FUNCTION "CWA_ScaleCtrlSub" : VOID	// FC 40
TITLE = CWA SUBROUTINE
//  
//COPYRIGHT:    (C) 1996 BY  BUHLER LTD.
//                           CH-9240 UZWIL  SWITZERLAND
//
//PRODUCT:      CWA
//
//TITLE:        SCALE CONTROL: SUBROUTINE
//
//-------------------------------------------------------------------------
//
//IDENT:        AUTOR:              DEPT:                         DATE:
//
//FC40.1.8      A. Egli             CT3                           27-Jun-2005
//              Working step: Do not calculate ingredient size 
//FC40.1.7      A. Egli             CT3                           21-Sep-2004
//              Registration: Test Ingr.WtActual >0 
//FC40.1.6      A. Egli             CT3                           12-Jun-2003
//              Test if more than 48 bins 
//FC40.1.5      A. Egli             CT3                           12-April-2000
//              Negativ CutoffWt >= 2* ParTolPosWt 
//FC40.1E       A. Egli             CT3                           12-Nov-98
//              Fault in SUBROUTINE EMPTYING_MONITORING 
//              Run closing delay only if scale is open
//FC40.1D       A. Egli             CT3                           24-Jun-98
//              Start part recipe
//              DBB52: First Ingredient
//              DBB53: Number of Ingredient
//FC40.1C       A. Egli             AEE61                         18-Mar-98
//              Update to S5 Version 2F
//
//FC40.1B       A. Egli             AEE61                         20-Jan-98
//              Update to S5 Version 2D
//
//FC40.1A       S. Kalberer         AEE61                         24-Apr-96
//              1st Release in S7, converted from FB40.1D
//
//-------------------------------------------------------------------------
//
//PURPOSE:      MANUAL : CWAMAN
//
//RESTRICTIONS:
//
//-------------------------------------------------------------------------
//
//$EJECT
//
AUTHOR : EA
FAMILY : CWA
NAME : CWASubr
VERSION : 1.8
VAR_TEMP
  InCode : WORD ;	//InFunctionCode
  TargetAddress : DWORD ;	//temp address pointer
  Cnt : WORD ;	//temp loop counter
  tmpAddr : DWORD ;
  tmpTimeTarget : INT ;
  tmpTimeTotal : INT ;
  tmpWtPartIngr : DINT ;
  tmpWtDiff : DINT ;
  tmpWtCorr : DINT ;
  tmpWt : DINT ;
  tmpBinNr : INT ;
  tmpWtDiffIsPos : BOOL ;
END_VAR
BEGIN
NETWORK
TITLE = FC-PARAMETER
//FC-PARAMETER:
//-------------
//  CODE: CODE OF EXECUTING FUNCTION
//        KY 0,0   : SUBROUTINE RESET TIMER
//        KY 0,1   : SUBROUTINE RUN DosingMonDelay
//        KY 0,2   : SUBROUTINE RUN SettlingTime
//        KY 0,4   : SUBROUTINE DOSING_MONITORING
//        KY 0,5   : SUBROUTINE EMPTYING_MONITORING
//        KY 0,8   : SUBROUTINE RUN DAMPENING TIME SCALE CLOSED
//        KY 0,10  : SUBROUTINE RUN CLOSING DELAY IF EMPTY
//        KY 0,11  : SUBROUTINE CORRECTION CUTOFF VALUE
//        KY 0,12  : SUBROUTINE TOLERANCE TEST
//                   Input : DW196 = var_tol._pos_unit
//                           DW197 = var_tol._pos_%
//                   Output: M199.0: 1=fault pos
//                   Output: M199.1: 1=fault neg
//                   Output: M199.2: 1=Ingr.Done
//        KY 1,1   : SUBROUTINE TEST_RESULT_DB
//        KY 1,2   : SUBROUTINE INIT_RESULT
//        KY 1,4   : SUBROUTINE REGISTRATION_INGREDIENT
//        KY 2,1   : SUBROUTINE TEST_RECIPE_DB
//        KY 2,2   : SUBROUTINE COUNT INGR
//        KY 2,4   : SUBROUTINE READ RECIPE INGR
//        KY 2,8   : SUBROUTINE MODIFY_RECIPE
//        KY 4,1   : SUBROUTINE TEST_BIN_PARAMETER_DB
//        KY 4,2   : SUBROUTINE READ_BIN_PARA
//        KY 4,4   : SUBROUTINE WRITE_BIN_PARA
//        KY 4,8   : SUBROUTINE TEST BIN
//                      Input  : DW195 = Bin-Nr
//                      Output : M 199.3 : 1= Fault
//                               DW197 = DW_NR_Bin
//                               DW198 = relBinNr
//
//ACTUAL DB BY CALL: SCALE    DB
//AUFGESCHALGENER  : WAAGEN   DB
//
//
      T     #InCode;
NETWORK
TITLE = Subroutine Reset Time
//Not implemented.
//Instead of this function call, write your self:
//      L     S5T#0MS                     // Partimer_1
//      SE    T [DBW 24]                  // --> Reset Timer
NETWORK
TITLE =  Subroutine Run DosingMonDelay
      L     #InCode;
      L     B#(0, 1);	// CODE= Run Settling time dos.
      <>I;
      JC    NX4;	// NEXT;
      AN    M 189.3;	// --> inf_DelayMon
      ON    "SYS_Tick1s";
      BEC;
      L     DBW 96;	// var_DosingMonDelay
      +     10;
      T     DBW 96;	// var_DosingMonDelay
      L     DBW 160;	// ParDosingMonDelay
      >=I;
      R     M 189.3;	// --> inf_DelayMon
      BEU;
NETWORK
TITLE =  Subroutine Run Settling time
NX4:  L     #InCode;
      L     B#(0, 2);	// CODE= Run Settling time
      <>I;
      JC    NX5;
      L     W#16#999;
      L     DBW 194;	// ParSettlingTime
      DTB;
      <D;
      JC    NX4s;
      L     W#16#1000;	// time_base 1/10s
NX4a: OW;
      A     M 193.4;	// --> sta_SettlingTime
      SD    T [DBW 24];	// Partimer_1 --> Timer
      A     T [DBW 24];	// Partimer_1 --> Timer
      R     M 193.4;	// --> sta_SettlingTime
      BEU;
NX4s: SRW   4;
      L     W#16#2000;	// time_base 1 s
      JU    NX4a;
NETWORK
TITLE =  Subroutine Dosing monitoring
NX5:  L     #InCode;
      L     B#(0, 4);	// CODE= dos_MONITORING
      <>I;
      JC    NX6;	// NEXT;
      L     DBW 378;	// var_MonTime
      L     0;
      >I;
      JC    OK5;	// -- INIT --------------------
      L     DBW 162;	// ParDosingMonTime
      T     DBW 378;	// --> var_MonTime
      L     DBD 254;	// inf_ScaleWt
      T     DBD 380;	// --> var_MonTara
OK5:  AN    "SYS_Tick1s";	// -- CONTROL -----------------
      BEC;
      A     M 191.2;	// es_DosingMon
      O     M 189.3;	// inf_DosingMon
      JC    TI2;
      L     DBW 378;	// var_MonTime [1/10s]
      +     -10;
      T     DBW 378;	// --> var_MonTime [1/10s]
      L     0;
      >I;
      JC    TI2;	// --- CONTROL ---------------
      L     DBW 166;	// ParDosingMonWtFast
      A     M 180.6;	// outp_DosingFast
      JC    X1;
      L     DBW 168;	// ParDosingMinWtSlow
X1:   L     DBD 380;	// var_MonTara
      A     DBX 7.0;	// ParNegativeWeighing
      JC    NX5n;
      +D;
      L     DBD 254;	// inf_ScaleWt
      >=D;
      AN    DBX 7.0;	// ParNegativeWeighing
      JC    ERRO;
      JU    TI2;
NX5n: TAK;
      -D;
      L     DBD 254;	// inf_ScaleWt
      <D;
      JC    ERRO;
      JU    TI2;
ERRO: S     M 191.2;	// --> es_time_outdos
      L     63;
      T     DBW 246;	// --> errCodeSW
TI2:  L     DBW 328;	// Ingr.DosingTime
      L     DBW 354;	// ParDosingTimeMax
      <=I;
      O(;
      L     0;	// no monitioring
      ==I;
      );
      BEC;	// --- error 2 -------------------
      S     M 191.4;	// --> es_DosingTime
      L     64;
      T     DBW 246;	// --> errCodeSW
      BEU;
NETWORK
TITLE =  Subroutine Emptying monitoring
NX6:  L     #InCode;
      L     B#(0, 5);	// CODE= Emptying monitoring
      <>I;
      JC    NX7;	// NEXT;
      L     DBW 378;	// var_MonTime
      L     0;
      >I;
      JC    OK6;	// -- INIT -------------------
      L     DBW 164;	// ParEmptyingMonTime
      T     DBW 378;	// --> var_MonTime [s]
      L     DBD 254;	// inf_ScaleWt
      T     DBD 380;	// --> var_MonTara
OK6:  AN    "SYS_Tick1s";	// -- CONTROL -----------------
      BEC;
      L     DBW 376;	// var_emptying_time
      +     1;
      T     DBW 376;	// --> var_emptying_time
      L     DBW 172;	// ParEmptyingTimeMax
      <=I;
      O(;
      L     0;	// no monitioring
      ==I;
      );
      JC    MONI;
      S     M 191.1;	// --> es_emptying_time
      L     62;
      T     DBW 246;	// --> errCodeSW
MONI: L     DBW 378;	// var_MonTime [1/10s]
      L     10;	//[1E]
      -I;
      T     DBW 378;	// --> var_MonTime [1/10s]
      JP    OUT;	// --- CONTROL ---------------
      L     DBD 380;	// var_MonTara
      L     DBW 170;	// ParEmptyingMonWt
      -D;
      L     DBD 254;	// inf_ScaleWt
      >=D;
      BEC;
      S     M 191.1;	// --> es_emptyingTime
      L     61;
      T     DBW 246;	// --> errCodeSW
OUT:  BEU;
NETWORK
TITLE =  Subroutine Run StartingDelay
NX7:  L     #InCode;
      L     B#(0, 8);	// CODE= Run StartingDelay
      <>I;
      JC    NX8;
      L     W#16#999;
      L     DBW 192;	// ParStartingDelay
      DTB;
      <D;
      JC    NX8s;
      L     W#16#1000;	// time_base 1/10s
NX8a: OW;
      A     M 193.7;	// sta_StartingDelay
      SD    T [DBW 24];	// Partimer_1 --> Timer
      A     T [DBW 24];	// Partimer_1 --> Timer
      R     M 193.7;	// --> sta_StartingDelay
      BEU;
NX8s: SRW   4;
      L     W#16#2000;	// time_base 1 s
      JU    NX8a;
NETWORK
TITLE =  Subroutine Run Closing Delay
NX8:  L     #InCode;
      L     B#(0, 10);	// CODE= Run Closing Delay
      <>I;
      JC    NX9;
      L     W#16#999;
      L     DBW 196;	// ParClosingDelay
      DTB;
      <D;
      JC    NX9s;
      L     W#16#1000;	// time_base 1/10s
NX9a: OW;
      A     M 193.5;	// sta_ClosingDelay
      A     M 182.6;	// inp_open [1E]
      SD    T [DBW 24];	// Partimer_1 --> Timer
      A     T [DBW 24];	// Partimer_1 --> Timer
      R     M 193.5;	// --> sta_ClosingDelay
      BEU;
NX9s: SRW   4;
      L     W#16#2000;	// time_base 1 s
      JU    NX9a;
NETWORK
TITLE =  Subroutine Correction Cutoff
//Correction switch over value:
//-----------------------------
// mode 1:  actual_switch_over_time < (Parswitch_over_time/4)
// mode 2:  actual_switch_over_time > (Parswitch_over_time/4)
//
// Implementation:
// ===============
// Sequence will go through loop twice:
// 1. Correction of pre cutoff value:
//     var_CutoffWt and var_SwitchOverWt will be optimized.
//     Function: after dosing stop, weight is not in tolerance
// 2. Correction of switch over weight:
//     var_SwitchOverWt will be optimized.
//     Function: fine feeding time is not the same as ParSwitchOverTime
NX9:  L     #InCode;
      L     B#(0, 11);	// CODE= Correction Cutoff Value
      <>I;
      JC    NX10;
      R     M 199.0;	// VAR_LOOP_Cnt
      L     DBW 346;	// ParCutoffWtCorrMax
      L     0;
      ==I;
      BEC;
      L     DBW 174;	// ParCorrFactorMax [%]
      L     100;	//   max 100%
      <=I;
      JC    OK9;
      T     DBW 174;	// -->ParCorrFactorMax [%]
      AN    DBX 338.7;	// ParSwitchOwerWt (sign)
      JC    OK9;
      L     0;
      T     DBW 338;	// ParSwitchOverWt
OK9:  L     DBD 254;	// inf_ScaleWt
      L     DBD 324;	// Ingr.PartWtTara
      AN    DBX 7.0;	// ParNegativeWeighing
      JC    POS0;
      TAK;
POS0: -D;
      T     #tmpWtPartIngr;
      L     DBD 320;	// Ingr.PartWtTarget
      -D;
      T     #tmpWtDiff;	// --> var_difference
LOOP: L     #tmpWtDiff;
      L     0;
      >=D;
      =     #tmpWtDiffIsPos;
      TAK;
      JC    POS;	// --> overweight
      -D;	// ) (Invert)
      L     DBW 178;	// ParDeadBandNeg
      JU    T1;
//-- Overweight ---
POS:  L     DBW 176;	// ParDeadBandPos
T1:   ITD;
      >D;
      JC    CR1;	// --> correction overweight
      JU    SWI;	// --> no correction cutoffvalue
CR1:  L     DBW 174;	// ParCorrFactorMac [%]
      DTR;
      L     #tmpWtDiff;	// var_difference
      DTR;
      *R;
      L     1.000000e+02;	// /100
      /R;
      RND;
MIN:  T     #tmpWtCorr;	// --> var_correctionWt
      L     0;
      <>D;
      JC    JL1;
      L     #tmpWtDiff;	// var_difference == 0
      ==D;
      JC    JL1;
      L     1;
      A     #tmpWtDiffIsPos;
      JC    MIN;
      L     L#-1;
      JU    MIN;
JL1:  L     #tmpWtCorr;
      A     M 192.0;	// sta_testWeighment
      JC    CR2;
      L     DBW 346;	// ParCutoffWtCorrMax
      >D;
      JC    MAXP;	// --> max correction if positive
      +D;
      JM    MAXM;	// --> max correction in negative
      JU    CR2;
MAXP: T     #tmpWtCorr;
      JU    CR2;	// var_correctionWt
MAXM: L     DBW 346;	// ParCutoffWtCorrMax
      L     -1;
      *I;
      T     #tmpWtCorr;	// var_correctionWt
CR2:  AN    #tmpWtDiffIsPos;
      A     M 189.5;	// cmd_NorCorrCutoffWt
      O     M 199.0;	// VAR_LOOP_Cnt
      JC    CR3;	// --> only switchOverWt
      L     DBW 340;	// ParCutoffWt
      ITD;
      L     #tmpWtCorr;	// var_correctionWt
      +D;
      T     DBW 340;	// --> ParCutoffWt
//=== Begrenzung Vorabschaltwert >=0
CR3:  A     DBX 7.3;	//Negative CutoffWt                  //[1.5]
      JC    CR3P;
      L     DBW 340;	// ParCutoffWt
      L     0;
      >=I;
      JC    CR3A;
      T     DBW 340;	// --> ParCutoffWt
      T     #tmpWtCorr;	// var_correctionWt
      JU    CR3A;
//=== Begrenzung Vorabschaltwert >= minus 2* positive Toleranz    //[-->1.5]
CR3P: L     DBW 342;	// ParTolPosWt
      L     DBW 344;	// ParTolNegWt
      +I;
      NEGI;
      L     DBW 340;	// ParCutoffWt
      <=I;
      JC    CR3A;
      TAK;
      T     DBW 340;	// --> ParCutoffWt
      -I;
      ITD;
//-- Correcon for Switch over weight:
//  := tmpWtCorr - (ParCutoffWt-Limit)
      L     #tmpWtCorr;	// var_correctionWt
      TAK;
      -D;
      T     #tmpWtCorr;	// var_correctionWt
//Ende Berenzung auf Positive Toleranz                              //[<--1.5]
CR3A: AN    #tmpWtDiffIsPos;
      O     M 199.0;	// VAR_LOOP_Cnt
      A     M 189.5;	// cmd_NorCorrCutoffWt
      JC    SWI;
      L     DBW 338;	// ParSwitchOverWt
      ITD;
      L     #tmpWtCorr;	// var_correctionWt
      +D;
      T     DBW 338;	// --> ParSwitchOverWt
      L     0;
      >D;
      JC    SWI;
      L     1;
      T     DBW 338;	// --> ParSwitchOverWt
SWI:  A     M 199.0;	// VAR_LOOP_Cnt (Loop 2)
      BEC;
      S     M 199.0;	// --> VAR_LOOP_Cnt
      L     DBW 348;	// ParDoisngTimeSlow
      L     DBW 350;	// ParSwitchOverTime_f/s
      +I;
      T     #tmpTimeTarget;
      SRW   2;	// / 4
      L     DBW 330;	// Ingr.SwitchOverTime
      <=I;
      JC    MOD2;	// --> correction mode 2
      L     DBW 376;	// dos_time_Part_ingr [1]
      +I;
      T     #tmpTimeTotal;
// 
      L     #tmpTimeTarget;
      L     DBW 330;	// Ingr.SwitchOverTime
      -I;
      DTR;	// [1/10s]
      L     #tmpTimeTotal;
      DTR;
      /R;
      L     1.000000e-01;
      *R;
      L     #tmpWtPartIngr;
CALC: DTR;
      *R;
      RND;
      T     #tmpWtDiff;	// --> var_difference
      JU    LOOP;	// -- Mode 2 --------------------
MOD2: L     #tmpTimeTarget;
      DTR;
      L     DBW 330;	// Ingr.SwitchOverTime
      DTR;	// / 4
      /R;
      L     1.000000e+00;
      -R;
      L     DBW 338;	// ParSwitchOverWt_F/S
      JU    CALC;
NETWORK
TITLE =  Subroutine Tolerance
NX10: L     #InCode;
      L     B#(0, 12);
      <>I;
      JC    NX11;
      R     M 199.0;	// --> fault_pos
      R     M 199.1;	// --> fault_neg
      R     M 199.2;	// --> ingr_done
      L     DBD 312;	// ingr.WtActual
      L     DBD 308;	// ingr.WtTarget
      -D;
      T     DBD 316;	// -->ingr.WtDiff
      JM    NEG;	// IF neg. goto NEG
      L     DBD 316;	// ingr.WtDiff
      L     DBW 392;	// BIN.ParTolPosWt
      >D;
      L     72;
      JC    FPOS;	// ->fault pos.
      JU    REL1;
NEG:  L     DBW 344;	// BIN.ParTolNegWt
      L     DBD 316;	// ingr.WtDiff
      +D;
      JM    NEG1;	// ->fault neg.
      L     DBW 358;	// BIN.ParTolNegPc (%)
      DTR;
      L     1.000000e-03;	// / 1000
      *R;
      L     DBD 308;	// ingr.WtTarget
      DTR;
      *R;
      RND;
      L     DBD 316;	// ingr.WtDiff
      +D;
      JM    NEG2;
      JU    DONE;	// --> ingr_done
REL1: L     DBW 394;	// BIN.ParTolPosPc (%)
      DTR;
      L     1.000000e-03;	// / 1000
      *R;
      L     DBD 308;	// ingr.WtTarget
      DTR;
      *R;
      RND;
      L     DBD 316;	// ingr.WtDiff
      <D;
      L     73;	// CODE: pos._tol._%
      JC    FPOS;	// --> fault_pos
DONE: SET;
      S     M 199.2;	// --> ingr_done
      BEU;
NEG1: L     70;	// CODE: neg._tol._abs.
      JU    FNEG;
NEG2: L     71;	// CODE: neg._tol.%
FNEG: AN    DBX 337.0;	// bin_type.ParmanualAdd
      O     M 193.3;	// StaPartIngr
      BEC;
      S     M 191.5;	// ->es_underWt
      S     M 199.1;	// ->fault_neg
      JU    FAUL;
FPOS: S     M 191.6;	// ->es_overWt
      S     M 199.0;	// ->fault_pos
FAUL: T     DBW 246;	// ->errCodeSW
      BEU;
NETWORK
TITLE =  Subroutine Test Result-DB
NX11: L     #InCode;
      L     B#(1, 0);	// CODE= For all Result-DB function
      AW;
      JZ    NX12;
      L     0;
      L     DBW 116;	// ParDBNrResultDB
      ==I;
      BEC;
      L     10;
      AN    DBX 9.4;	// ParResultRecFull
      JC    CE1;
      L     16;
CE1:  L     DBW 122;	// ParNoOfBytePerRecord
      >I;
      JC    ERR3;	// --> record to small
      L     DBW 120;	// ParNoOfRecords
      L     DBW 122;	// ParNrOfBytePerRecord
      *I;
      L     DBW 118;	// ParDW_NrResult
      +I;
      +     18;	// len_header
      T     DBW 392;	// --> var_target_len (WORD)
      OPN   DI [DBW 116];	// ParDB_NrResult
      L     DILG;	// length DB (in BYTE)
      T     DBW 394;	// --> var_DB_length
      L     DBW 392;	// --> var_target_len
      <I;
      JC    ERR2;
      L     DBW 118;	// ParByteNrResult
      SLD   3;	// bit-offset
      LAR2;
      L     B#(1, 1);
      L     #InCode;	// CODE= Test_Result_DB
      ==I;
      BEC;
      JU    NX12;
ERR3: L     55;	// --> record to small
      JU    ERR;
ERR2: L     54;	// --> result_DB to small
ERR:  S     DBX 3.3;	// --> cfg_fault_RESULT
      S     M 190.4;	// --> es_cfg_SPS
      T     DBW 246;	// --> errCodeSW
      BEU;
NETWORK
TITLE =  Subroutine Init_result_DB
NX12: L     #InCode;
      L     B#(1, 2);	// CODE= INIT_RESULT_DB
      <>I;
      JC    NX13;	// NEXT;
      L     DBD 258;	// job number
      T     DID [AR2,P#0.0];	// --> R_DB.job_number
      L     DBD 262;	// recipe_nr / batch_nr
      T     DID [AR2,P#4.0];	// --> R_DB.recipe_nr /batch_nr
      L     2#0;
      T     DIW [AR2,P#8.0];	// --> R_DB.status_result
      L     0;
      T     DID [AR2,P#10.0];	// --> R_DB.TotalWtTarget
      T     DID [AR2,P#14.0];	// --> R_DB.TotalWtActual
      +AR2  P#18.0;
      L     DBW 120;	// ParNrOfRecords
      L     DBW 122;	// ParNrOfByPerRecord
      *I;
      SRW   1;
LP12: T     DBW 394;	// --> var_NrOfDWClear
      L     0;
      <=I;
      BEC;
      T     DIW [AR2,P#0.0];	// save result
      +AR2  P#2.0;	// set pointer to next DW 
      L     DBW 394;	// Var_NrOfDW_clear
      +     -1;
      JU    LP12;	// LOOP;
NETWORK
TITLE =  Subroutine Registration Ingredient
NX13: L     #InCode;
      L     B#(1, 4);	// CODE= REGISTRATION_INGREDIENT
      <>I;
      JC    NX14;	// NEXT;
      TAR2;	// <-- ADDRESS-RESULT-DB (first DW)
      T     #tmpAddr;	// --> var_address_header
      L     DBD 312;	//[1.7] Ingr.WtActual
      L     0;	//[1.7]
      >=D;	//[1.7]
      JC    X13P;	//[1.7]
      T     DBD 312;	//[1.7]
X13P: AN    M 193.2;	// sta_singleIngrAc
      JC    J1;
      L     DIW [AR2,P#8.0];	// R_DB.statusResult
      L     2#1;	// sta_withModif
      OW;
      T     DIW [AR2,P#8.0];	// --> R_DB.statusResult
J1:   L     DBD 312;	// Ingr.WtActual
      A     M 188.3;	// cmd_ModifReady
      JC    X01;
      L     DBD 308;	// Ingr.WtTarget
X01:  T     #tmpWt;
      L     DID [AR2,P#10.0];	// R_DB.TotalWtTarget
      +D;
      T     DID [AR2,P#10.0];	// --> R_DB.TotalWtTarget
      L     DBD 312;	// Ingr.WtActual
      L     DID [AR2,P#14.0];	// R_DB.TotalWtActual
      +D;
      T     DID [AR2,P#14.0];	// --> R_DB.TotalWtActual
      L     #tmpWt;
      L     DBD 274;	// TotalWtTarget
      +D;
      T     DBD 274;	// TotalWtTarget
      L     DBD 312;	// Ingr.WtActual
      L     DBD 278;	// TotalWtActual
      +D;
      T     DBD 278;	// TotalWtActual
      +AR2  P#18.0;	// - Startadress search Bin -----
      L     0;
      T     #tmpBinNr;	// -->var_bin_nr
      AN    DBX 9.2;	// ParResultRecPerBin
      JC    FIND;
      L     DBW 306;	// ingr.bin_nr
      T     #tmpBinNr;
      AN    DBX 9.3;	// ParResultRecSorted
      JC    FIND;
      L     DBW 332;	// ingr.RelBinNr
      L     DBW 120;	// ParNrOfrecords
      >=I;
      BEC;	// --> no bin
      L     DBW 332;	// ingr.RelBinNr
      L     DBW 122;	// ParNrOfByPerRecord
      *I;
      SLD   3;	// bit-offset
      +AR2;	// --> AdrNextIngr
      JU    SAVE;
FIND: L     0;	// --- search record -------------
LP13: T     #Cnt;
      L     DBW 120;	// ParNrOfrecords
      >=I;
      JC    ER13;	// ER13;
      L     0;
      L     DIW [AR2,P#0.0];	// --> last Ingredient
      ==I;
      O(;
      L     #tmpBinNr;	// -->var_bin_nr
      ==I;
      );
      JC    SAVE;
      L     DBW 122;	// ParNrOfByPerRecord
      SLD   3;	// bit-offset
      +AR2;	// --> adr_next_ingr
      L     #Cnt;	// var_record_Cnt
      +     1;
      JU    LP13;	// LOOP;
//--- SAVE ------------------------
SAVE: L     DBW 306;	// ingr.bin_nr
      T     DIW [AR2,P#0.0];	// --> bin_nr
      L     #tmpWt;	// Ingr.WtActual
      L     DID [AR2,P#2.0];	// REG_DB.value_target
      +D;
      T     DID [AR2,P#2.0];	// --> REG_DB.TotalWtTarget
      L     DBD 312;	// Ingr.WtActual
      L     DID [AR2,P#6.0];	// R_DB.TotalWtActual
      +D;
      T     DID [AR2,P#6.0];	// --> REG_DB.TotalWtActual
      AN    DBX 9.4;	// ParResultRecFull
      BEC;
      L     DBW 328;	// dos_time
      L     DIW [AR2,P#10.0];	// REG_DB.dos_time
      +D;
      T     DIW [AR2,P#10.0];	// --> REG_DB.dos_time
      L     DBD 338;	// BIN.SwitchOverWt_F/S.var_CutoffWt
      T     DID [AR2,P#12.0];	// --> REG_DB.SwitchOverWt_F/S.var_CutoffWt
      BEU;
ER13: L     74;	// --> Code: Result-DB full
      T     DBW 246;	// --> errCodeSW
      LAR2  #tmpAddr;	// Var_address_header
      SET;
      S     DIX [AR2,P#9.1];	//R_DB.Status.OutOfMemory
      BEU;
NETWORK
TITLE =  Subroutine Test Recipe-DB
NX14: L     #InCode;
      L     B#(2, 0);	// CODE=for all recipe-DB function
      AW;
      JZ    NX15;	// NEXT;
      L     DBW 104;	// ParNrOfingr
      L     DBW 106;	// ParNrOfByPerIngr
      *I;
      L     DBW 102;	// ParNrOfrecipe
      *I;
      L     DBW 100;	// ParDW_NrFirstRecipe
      +I;
      T     DBW 392;	// --> var_NrOfByForDB
      OPN   DI [DBW 98];	// ParDB_Nr_recipe
      L     DILG;	// length DB (in BYTE)
      L     DBW 392;	// var_NrOfByForDB
      <I;
      JC    ER14;	// --> recipe_DB to small
      L     #InCode;
      L     B#(2, 1);	// CODE= Test_Recipe_DB
      ==I;
      BEC;
      L     DBW 104;	// ParNrOfingr
      L     DBW 106;	// ParNrOfDW/ingr
      *I;
      L     DBW 70;	// inf_recipe_place
      *I;
      L     DBW 100;	// ParDWNRFirstRecipe
      +I;	// --> var_first_DW_active_recipe
      SLD   3;	// bit-offset
      LAR2;	// --> bit-adr: VarFirstDWActiveRecipe
      JU    NX15;	// NEXT;
ER14: L     52;	// --> errCodeSW
      T     DBW 246;	// --> CfgFaultRecipeDB
      S     DBX 3.1;	// --> err_cfg_fault_SPS
      S     M 190.4;
      BEU;
NETWORK
TITLE =  Subroutine Count Component
NX15: L     #InCode;
      L     B#(2, 2);	// CODE= Count ingr
      <>I;
      JC    NX16;	// NEXT;
      L     0;
LP15: T     DBW 294;	// IngrCntTotal
      L     DBB 52;	// Offset Ingr
      +I;
      L     DBW 104;	// ParNrOfingr
      >=I;
      BEC;
      L     0;
      L     DIW [AR2,P#0.0];	// --> last ingredient
      ==I;
      BEC;
      L     0;
      L     DBB 53;	//Number of part ingredient
      <>I;
      A(;
      L     DBW 294;	//IngrCntTotal
      L     DBB 53;	//Number of part ingredient
      >=I;
      );
      BEC;
      L     DBW 106;	// ParNrOfByPerIngr
      SLD   3;	// bit-offset
      +AR2;	// --> adr_next_ingr
      L     DBW 294;	// IngrCntTotal
      +     1;
      JU    LP15;	// LOOP;
NETWORK
TITLE =  Subroutine Read Recipe Component
NX16: L     #InCode;
      L     B#(2, 4);	// CODE= Read Recipe_ingr
      <>I;
      JC    NX17;	// NEXT;
      L     DBW 292;	// IngrCnt (actual)
      L     DBB 52;	// Offset Ingr
      +I;
      L     DBW 104;	// ParNrOfingr
      >I;
      JC    EMPT;	// --> Emptying scale
      L     0;
      L     DBB 53;	//Number of part ingredient
      <>I;
      A(;
      L     DBW 292;	//IngrCnt (actual)
      L     DBB 53;	//Number of part ingredient
      >I;
      );
      JC    EMPT;	// --> Emptying scale
      L     DBW 292;	// IngrCnt (actual)
      L     DBB 52;	// Offset Ingr
      +I;
      +     -1;
      L     DBW 106;	// ParNrOfByPerIngr
      *I;
      SLD   3;	// bit-offset
      +AR2;	// --> adr_ingr
      L     DIW [AR2,P#0.0];
      T     DBW 306;	// --> ingr_bin_nr
      L     0;	//[1.8]
      <=I;	//[1.8]
      L     DID [AR2,P#2.0];	// ingr.target_weight
      JC    DIFF;	//[1.8]
      AN    DBX 7.5;	// ParIngrSizePc
      JC    JL16;
      DTR;
      L     1.000001e-04;	// * 0.0001
      *R;
      L     DBD 270;	// batch_size_recipe
      DTR;
      *R;
      RND;
JL16: AN    DBX 7.4;	// ParBatchSizePc
      JC    DIFF;
      DTR;
      L     DBW 268;	// batch_size_%%
      DTR;
      *R;
      L     1.000001e-03;	// * 0.001
      *R;
      RND;
DIFF: T     DBD 308;	// --> ingr_target_value
      L     0;
      T     DBD 312;	// --> ingr.WtActual
      TAK;
      -D;
      T     DBD 316;	// --> ingr.WtDiff
      BEU;
EMPT: L     0;
      T     DBW 306;	// --> ingr_bin_nr
      T     DBD 308;	// --> ingr_target_value
      BEU;
NETWORK
TITLE =  Subroutine Modify Bin in Recipe
NX17: L     B#(2, 8);	// CODE= Modify Recipe
      L     #InCode;
      <>I;
      JC    NX18;
      L     0;
LP17: T     #Cnt;	// IngrCntTotal
      L     DBW 104;	// ParNrOfingr
      >=I;
      BEC;
      L     DBW 306;	// ingr.bin_nr
      L     DIW [AR2,P#0.0];	// --> last ingredient
      <>I;
      JC    INKR;
      L     DBW 90;	// VarPreselectedBin
      T     DIW [AR2,P#0.0];	// --> recipe.bin_nr
INKR: L     DBW 106;	// ParNrOfByPerIngr
      SLD   3;	// bit-offset
      +AR2;	// --> adr_next_ingr
      L     #Cnt;	// IngrCntTotal
      +     1;
      JU    LP17;
NETWORK
TITLE =  Subroutine Test Bin_Parameter_DB
NX18: L     #InCode;
      L     B#(4, 0);	// CODE=for all BIN-DB function
      AW;
      JZ    NX19;	// NEXT;
      L     DBW 108;	// ParDB_NR_Bin_Data
      L     0;
      ==I;
      BEC;	// --> no bin_data_DB
      L     DBW 114;	// ParNrOfByPerBin
      L     42;
      <I;
      JC    OK1;
      T     DBW 114;	// --> ParNrOfByPerBin
OK1:  L     DBW 112;	// ParNrOfbin
      L     DBW 114;	// ParNrOfByPerBin
      *I;
      L     DBW 110;	// ParDWNRFirst_bin
      +I;
      T     DBW 392;	// --> var_NrOfDW
      OPN   DI [DBW 108];	// ParDB_Nr_Bin_Data
      L     DILG;	// length DB (in BYTE) 
      L     DBW 392;
      <I;
      JC    ER18;	// --> recipe_DB to small
      L     #InCode;
      L     B#(4, 1);	// CODE= Test_Bin_DB
      ==I;
      BEC;
      JU    NX19;	// --> OK; NEXT;
ER18: L     57;	// CODE:bin_data_DB to samll
      T     DBW 246;	// --> errCodeSW
      S     DBX 3.2;	// --> cfgFaultBinDataDB
      S     M 190.4;	// --> err_cfg_fault_SPS
      S     M 199.3;	// --> Output Fault
      BEU;
NETWORK
TITLE =  Subroutine Bin's
NX19: L     #InCode;
      T     MB 199;
      L     B#(4, 0);	// CODE=for all BIN-DB function
      AW;
      JZ    NX20;	// NEXT;
      R     M 190.3;	// --> err_illegel_ingr
      A     M 199.0;	// Test Bin-DB
      BEC;
      L     DBW 306;	// ingr.bin_nr
      L     0;	// NO_BIN
      <=I;
      AN    M 199.3;	// Mode =Test Bin
      BEC;
      L     DBW 390;	// var_preselected_bin
      L     0;	// NO_BIN
      <=I;
      A     M 199.3;	// Mode =Test Bin
      JC    OK_F;
      L     DBW 110;	// ParDWNrFirstBin
      SLD   3;	// bit-offset
      LAR2;	// --> adr_first_bin
      L     DBW 110;	// ParDWNrFirstBin
      T     DBW 394;	// --> var_DW_nr_read
      L     0;
LP19: T     DBW 396;	// ingr.RelBinNr
      L     DBW 112;	// ParNrOfbin
      >=I;
      JC    ER19;	// --> bin not found
      L     DBW 306;	// ingr.bin_nr
      L     DIW [AR2,P#0.0];	// bin_DB.nin_nr
      ==I;
      AN    M 199.3;	// MODE =TEST_BIN
      JC    READ;
      L     DBW 390;	// var_preselected_bin
      ==I;
      A     M 199.3;	// MODE =TEST_BIN
      JC    OK_F;	//OK-F;
      L     DBW 114;	// ParNrOfDW/bin
      SLD   3;	// bit-offset
      +AR2;	// --> adr_next_bin
      L     DBW 394;	// var_DW_nr_read
      L     DBW 114;	// ParNrOfByPerBin
      +I;
      T     DBW 394;	// --> var_ByNrRead
      L     DBW 396;	// ingr.RelBinNr
      +     1;
      JU    LP19;	// 
READ: L     DBW 396;	// var_relBinNr
      T     DBW 332;	// ingr.RelBinNr
      A     M 199.2;	// MODE =WRITE
      JC    WRIT;
//--Copy parameter to scale-DB --------
      L     P#334.0;
      T     #TargetAddress;	// --> VarDWNrTarget
      L     DBW 394;	// VarDWNrRead
      SLD   3;	// bit-offset
      LAR2;	// var_DWNrSource --> AR2
      L     DBW 114;	// ParNrOfBytePerBin
COLP: T     #Cnt;	// LOOP Counter
      L     DIB [AR2,P#0.0];
      T     DBB [#TargetAddress];	// Scale-DB
      +AR2  P#1.0;	// INC SourceAddress (2 Byte)
      L     #TargetAddress;	// INC TargetAddress (1 Word)
      +     L#8;
      T     #TargetAddress;
      L     #Cnt;	// LOOP Counter
      LOOP  COLP;	// COPY-LOOP
      L     0;
      T     DBD 46;
      T     DBW 50;	//--> activeBin[xx..1]
      L     48;
      L     DBB 333;	// ingr.RelBinNr
      <=I;
      BEC;	//[1.6]
      LAR1;
      S     DBX [AR1,P#46.0];	//-->ActiveBin[x]
      BEU;
ER19: L     58;	// CODE: bin not found
      T     DBW 246;	// --> errCodeSW
      AN    M 199.3;	// MODE= Test_Bin
      S     M 190.3;	// --> err_illegal_ingr
      BEU;
WRIT: L     DBW 114;	// ParNrOfByPerBin
      L     8;
      <I;
      BEC;
      L     DBD 338;	// var_switchOver/var_cutoffWt
      T     DID [AR2,P#4.0];	// --> Store
      BEU;
OK_F: R     M 199.3;	// Mode= Test_Bin
      BEU;
NETWORK
TITLE =
NX20: BE;
END_FUNCTION

FUNCTION "CWA_ScaleCtrlMain" : VOID	// FC 41
TITLE = CWA SCALE-MAIN
//
//COPYRIGHT:    (C) 1996  BUHLER AG, CH-9240 UZWIL, SWITZERLAND
//
//PRODUCT:      GCS7 - CWA 32 Bit
//
//TITLE:        SCALE CONTROL: MAIN PROGRAM
//
//-------------------------------------------------------------------------
//
//IDENT:        AUTHOR:             DEPT:                       DATE:
//
//FC41.2.9      A.Egli              CT3                         02-Apr-2009
//                -Do not convert CmdAcceptWeight to CmdAbortIngr if ErrZeroTol
//FC41.2.8      A.Egli              CT3                         02-Mai-2005
//                  Calculation speed when change fast to slow 
//                  DBX81.3: temporare flag, to store event "New ingredient"
//FC41.2.7      A.Egli              CT3                         02-Jul-2004
//                  Do not calculate Ingr.WtActual during deselect bin
//FC41.2.6      A.Egli              CT3                         02-Jul-2004
//                  Step: 5500: Reset inf_FlagStopValue when new ingredient
//                  Because interrupt OB can set this in the meantime             
//FC41.2.5      A.Egli              CT3                         04-Mar-2004
//                  CmdRestDischargeOff
//FC41.2.4      A.Egli              CT3                         27-Mar-2004
//                  StatePC= 4002 when StateSW=Hex3000
//FC41.2.3      A.Egli              CT3                         18-Nov-2003
//                  Start as Single Ingredient: Reset Total
//FC41.2.2      A.Egli              CT3                         15-Jan-2003
//              Change to tipping, 
//                  if rest-weight < switch over weight fast slow
//FC41.2.1      A.Egli              CT3                         14-Oct-2002
//              Offline check if Hsk are set
//FC41.2.0      A.Egli              CT3                         11-Oct-2001
//              PC Direct Control Interface  
//FC41.1.11     A.Egli              CT3                         26-Jan-2001
//              Only reset WtScale if ParPulseXxxCall 
//FC41.1.10     S. Kalberer         CT3                         31-Oct-2000
//              Update to S5.2K: At change to interm.Dischar. sta_reconveying
//FC41.1.9      A. Egli             CT3                         22-Jul-2000
//              Clear DBD254 if no emptying step
//FC41.1.8      A. Egli             CT3                         25-Apr-2000
//              Log message TipPulse with wrong parameter
//FC41.1H       A. Egli             CT3                         23-Mar-1999
//              Manual Addition: Accept under weight in state 5120 
//FC41.1G       A. Egli             CT3                         05-Mar-1999
//              Clear BinNr by reset and CmdAbortBatch 
//              Manual Addition: Alarm reset in state 5120 befor CmdManAddReady
//FC41.1F       A. Egli             CT3                         12-Nov-1998
//              Update to S5.2I: Abort batch in state Intermediate discharge 
//FC41.1E       A. Egli             CT3                         02-Nov-1998
//              Update to S5.2H: Clear counter var_reconveying at refill 
//FC41.1D       A. Egli             AEE61                       18-Mar-1998
//              Update to S5.2H 
//FC41.1C       A. Egli             AEE61                       16-Jan-1998
//              Update to S5.2G 
//FC41.1B       A. Egli             AEE61                       15-Aug-1997
//              Update to S5.2E
//FC41.1A       A. Egli             AEE61                       25-Apr-1996
//              1st Release, converted from S5.FB41.1K
//
//-------------------------------------------------------------------------
//
//PURPOSE:      MANUAL : CWAMAN
//
//RESTRICTIONS: USED FLAGS MW180-255
//
//-------------------------------------------------------------------------
//
AUTHOR : EA
FAMILY : CWA
NAME : CWAMain
VERSION : 2.9
VAR_TEMP
  tmpStoreAR2 : DINT ;
  tmpValue : DINT ;
  tmpStopFlag : BOOL ;
  tmpWord : INT ;
  tmpFlags : WORD ;
  tmpSpeed : INT ;
  tmpTimer : INT ;
  tmpBit : INT ;
  tmpFlagShift : INT ;
  tmpDBSource : INT ;
  tmpDWSource : INT ;
  tmpDBDestination : INT ;
  tmpDWDestination : INT ;
  tmpLenCopy : INT ;
  tmpFault : BOOL ;
  tmpScaleDB : INT ;
  tmpScalePara : BOOL ;
  tmpBinPara : BOOL ;
  tmpNewIngr : BOOL ;
END_VAR
BEGIN
NETWORK
TITLE = FC-PARAMETER
//
//ACTUAL DB BY CALL: SCALE DB
//
      L     DBNO;
      T     #tmpScaleDB;
      TAR2  #tmpStoreAR2;	// Store AR2
      CLR;	//[2.6]
      =     #tmpNewIngr;	//[2.6]
NETWORK
TITLE = PC Direct Contrl
      L     DBW 28;	//ScaleDB.ParScaleNr
      L     "SYS_DirectCtrlDB".PC.ObjectNo;	// DB3.ObjectNr
      <>I;	// 
      JC    DCEn;
      L     0;	//  )
      L     "SYS_DirectCtrlDB".PC.Hsk;	//  ) DB3.handshake_PC_GC
      ==I;	//  )
      JC    DCEn;	//  )
      L     3103;	// )  scale_parameter
      L     "SYS_DirectCtrlDB".PC.ObjectType;	// )  DB3.object_type
      ==I;	// )
      =     #tmpScalePara;
      L     3104;	// )  bin_parameter
      ==I;	// )
      =     #tmpBinPara;
      AN    #tmpScalePara;
      AN    #tmpBinPara;
      JC    DCEn;	// 
//Scale Parameter Init =========
      L     58;
      T     #tmpDWSource;
//Bin Parameter Init =========
      AN    #tmpBinPara;
      JC    DCSc;
      L     "SYS_DirectCtrlDB".PC.Value[1];	// )   DB3.bin_number
      OPN   DB [#tmpScaleDB];	// >>  CALL scale_DB
      T     DBW 390;	// --> Input FB40.VarBinNr
      L     W#16#408;
      UC    "CWA_ScaleCtrlSub";	// CWA.Subroutine Test Bin
      A     M 199.3;	//  )  error
      L     DBW 246;	//  )  CWA.errCodeSW
      JC    DCEr;	//  )=>bin_not_found
      L     DBW 394;	// Output.VarDWnr
      T     #tmpDWDestination;
      L     DBW 108;	// SCDB.ParDBNrBinData
      T     #tmpDBDestination;
      L     DBW 114;	// SCDB.ParNrOfBytePerBin
      T     #tmpLenCopy;
      JU    DCMv;
// ====Scale Parameter============
DCSc: L     #tmpScaleDB;
      T     #tmpDBDestination;
      L     160;
      T     #tmpDWDestination;
      L     46;
      T     #tmpLenCopy;
DCMv: A     "SYS_DirectCtrlDB".PC.Hsk.FDefinePara;	// F_DefinePara
      JC    DCPa;
      A     "SYS_DirectCtrlDB".PC.Hsk.FDefineCmd;	// F_DefineCmd
      JC    DCCd;
      JU    DCEx;
// ----- F_Define ---------------
DCCd: A     #tmpBinPara;
      JC    DCOK;
      AN    "SYS_DirectCtrlDB".PC.Cmd1[8];	// Cmd1.cmd_startSingleIngr
      AN    "SYS_DirectCtrlDB".PC.Cmd1[9];	// Cmd1.cmd_modifyBin
      JC    DCc2;
// -- Test new Bin --------------
      L     "SYS_DirectCtrlDB".PC.Value[1];	// DB3.bin_number
      OPN   DB [#tmpScaleDB];	// >>  CALL scale_DB
      T     DBW 390;	// --> Input FB40.var_bin_nr
      L     "SYS_DirectCtrlDB".PC.Value[1];	// )   DB3.bin_number
      OPN   DB [#tmpScaleDB];	// >>  CALL scale_DB
      T     DBW 390;	// --> Input FB40.var_bin_nr
      L     W#16#408;
      UC    "CWA_ScaleCtrlSub";	// CWA.Subroutine Test Bin
      A     M 199.3;	// error
      L     DBW 246;	// CWA.errCodeSW
      JC    DCEr;	// =>bin_not_found
//-- 
      AN    "SYS_DirectCtrlDB".PC.Cmd1[8];	// Cmd1.cmd_startSingleIngr
      OPN   DB [#tmpScaleDB];	// >>  CALL scale_DB
      JC    DCMO;
      A     DBX 251.0;	// sta_SingleIngrReq
      AN    DBX 78.2;	// cmd_SingleIngrReady
      AN    DBX 78.3;	// cmd_ModReady
      S     DBX 78.2;	// cmd_SingleIngrReady
      JC    DCCP;
      L     46;	// err: not ready for next
      JU    DCEr;
DCMO: S     DBX 78.3;	// ->cmd_ModReady
DCCP: L     "SYS_DirectCtrlDB".PC.Value[1];	// DB3.Inf_BinPreselected
      OPN   DB [#tmpScaleDB];	// >>  CALL scale_DB
      T     DBW 90;	// ->BinPreselected
      L     DB3.DBD 60;	// DB3.TargetValue
      OPN   DB [#tmpScaleDB];	// >>  CALL scale_DB
      T     DBD 92;	// ->TargetValue
DCc2: L     DB3.DBD 52;	// Cmd1/Cmd2
      OPN   DB [#tmpScaleDB];	// >>  CALL scale_DB
      L     2#11111111111111001111111111111111;	//[1E]
      AD;
      L     DBD 58;
      OD;
      T     DBD 58;	// --> function[47..32]
      L     "SYS_DirectCtrlDB".PC.Cmd3;	// CMD3
      OPN   DB [#tmpScaleDB];	// >>  CALL scale_DB
      L     DBW 62;
      OW;
      T     DBW 62;	// --> function[15..00]
      JU    DCOK;
      L     43;	// err_cfg_binlist
      JU    DCEr;
// ====Block Move  ================
DCPa: AN    #tmpBinPara;
      JC    fBIN;
      L     #tmpDWSource;
      +     4;
      T     #tmpDWSource;
      L     #tmpDWDestination;
      +     4;
      T     #tmpDWDestination;
      L     #tmpLenCopy;
      +     -4;
      T     #tmpLenCopy;
fBIN: NOP   0;
      CALL  "SYS_Copy_DBtoDB" (
           DBSource                 := 3,
           ByteSource               := #tmpDWSource,
           DBDest                   := #tmpDBDestination,
           ByteDest                 := #tmpDWDestination,
           NoOfByte                 := #tmpLenCopy,
           Fault                    := #tmpFault);
      JU    DCOK;
// ---- F_examine ----------------
DCEx: NOP   0;
      CALL  "SYS_Copy_DBtoDB" (
           DBSource                 := #tmpDBDestination,
           ByteSource               := #tmpDWDestination,
           DBDest                   := 3,
           ByteDest                 := #tmpDWSource,
           NoOfByte                 := #tmpLenCopy,
           Fault                    := #tmpFault);
DCOK: L     0;	// err_code
DCEr: T     "SYS_DirectCtrlDB".PC.ErrCode;	// ->DB3.error_code
      L     0;	// 
      T     "SYS_DirectCtrlDB".PC.Hsk;	// ->DB3.handshake_PC_GC
      SET;	// 
      S     "SYS_DirectCtrlDB".ChangeBit.CBit1;	// ->DB3.change-bit
DCEn: OPN   DB [#tmpScaleDB];
NETWORK
TITLE =  READ FLAGS
//
//MW 180 : COPY DW 21
//MW 182 :      DW 27
//MW 184 :      DW 28
//MW 186 :      DW 29
//MW 188 :      DW 39
//MW 190 :      DW 122
//MW 192 :      DW 124
//MW 194 :      DW 125
//MW 196 :      DW 126
      L     DBW 42;	// CommandsSSWtoUser
      T     MW 180;
      L     DBD 54;	// CommandsUserToSSW
      T     MD 182;
      L     DBW 58;	// function[47..32]
      T     MW 186;
      L     DBW 78;	// Internal flags
      T     MW 188;
      L     DBW 244;	// fault [15..00]
      T     MW 190;
      L     DBD 248;	// status[47..16]
      T     MD 192;
      L     DBW 252;	// status[15..00]
      T     MW 196;
NETWORK
TITLE =  O_SCALE
      L     0;
      L     DBW 208;	// handshakePCtoPLC
      ==I;
      JC    NX04;	// NEXT;
      S     DBX 207.1;	// --> cmd_interface_free
      L     W#16#F00;	// Q_Status...Q_Log_c.done
      AW;
      T     #tmpFlags;
      L     DBW 44;
      OW;
      T     DBW 44;	// --> cmd_xxx_done
      L     #tmpFlags;
      INVI;
      L     DBW 232;	// handshakePLCtoPC
      AW;
      T     DBW 232;	// --> handshakePLCtoPC
      L     0;
      T     DBW 236;	// --> errCodeAnswer
      AN    DBX 209.0;	// F_Define
      JC    QUIT;
      AN    DBX 211.0;	// cmd_startSingleIngr
      AN    DBX 211.1;	// cmd_modifyBin
      JC    CMD;
      L     DBW 218;	// inf_BinPreselected
      T     DBW 390;	// --> VAR_BinPreselected
      L     W#16#408;
      UC    "CWA_ScaleCtrlSub";	// S.Test Bin
      A     M 199.3;	// fault
      L     30;	// err: bin not found
      JC    ERRO;
      AN    DBX 211.0;	// cmd_startSingleIngr
      JC    MODI;
      A     M 195.0;	// sta_SingleIngrReq
      AN    M 188.2;	// cmd_SingleIngrReady
      AN    M 188.3;	// cmd_ModReady
      S     M 188.2;	// cmd_SingleIngrReady
      JC    COPY;
      L     46;	// err: not ready for i.c.
      JU    ERRO;
MODI: L     DBW 306;	// ingr.BinNr
      L     DBW 216;	// inf_deselected_bin
      <>I;
      A(;
      L     0;
      <>I;
      );
      L     45;	// err: bin not active
      JC    ERRO;
      AN    M 188.2;	// cmd_SingleIngrReady
      AN    M 188.3;	// cmd_ModReady
      S     M 188.3;	// --> cmd_ModReady
      JC    COPY;
      L     47;	// err: bin not active
ERRO: T     DBW 236;	// --> errCodeAnswer
      JU    CMD;
COPY: L     DBW 218;	// inf_BinPreselected
      T     DBW 90;	// --> BinPreselected
      L     DBD 220;	// TargetValue
      T     DBD 92;	// --> TargetValue
CMD:  L     DBW 210;	// FC[47..32]
      L     2#1111111111111100;
      AW;
      L     MW 186;	// FC[47..32]
      OW;
      T     MW 186;	// FC[47..32]
      L     DBW 212;	// FC[31..16]
      L     DBW 60;	// FC[31..16]
      OW;
      T     DBW 60;	// FC[31..01]
      L     DBW 214;	// FC[15..16]
      L     DBW 62;	// FC[15..00]
      OW;
      T     DBW 62;	// FC[15..00]
QUIT: L     0;
      T     DBW 208;	// handshakePCtoPLC
NETWORK
TITLE =  COMMANDS ASW
NX04: L     2#111111111;	//[2.5]
      L     DBW 60;	// FC[31..16]
      AW;
      INVI;
      L     MW 196;	// status[15..0]
      AW;
      T     MW 196;	// --> status[15..0]
      L     2#1111111000000000;	//[2.5]
      L     DBW 60;	// FC[31..16]
      AW;
      T     DBW 60;	// --> FC[31..16]
      L     2#1111111111;
      L     DBW 62;	// FC[15..0]
      AW;
      L     MW 196;	// status[15..0]
      OW;
      T     MW 196;	// --> status[15..0]
      L     2#1111110000000000;
      L     DBW 62;	// FC[15..0]
      AW;
      T     DBW 62;	// --> FC[15..0]
      L     W#16#F00;
      L     DBW 8;	// par_set_xx
      AW;
      L     MW 184;
      OW;
      T     MW 184;	// --> ASW.cmd_xx
      A     M 188.3;	// cmd_ModificationReady
      O     M 188.2;	// cmd_SingleIngrReady
      JC    NX05;	// NEXT;
      A     M 187.1;	// cmd_ModifyBin
      S     M 188.3;	// --> cmd_ModificationReady
      JC    CPY;	// COPY;
      AN    M 187.0;	// cmd_SingleIngr
      JC    NX05;	// NEXT;
      S     M 188.2;	// --> cmd_SingleIngrReady
CPY:  L     DBW 64;	// IngrNext.BinNr
      T     DBW 90;	// --> BinPreselected
      L     DBD 66;	// TargetValue
      T     DBD 92;	// --> TargetValue
NETWORK
TITLE =  OFF-LINE
//--> 
NX05: AN    M 183.7;	//ToASW.InfOffline
      JC    NX06;	// 
      L     2#111100000000;
      L     DBW 232;	//PCRead.Hsk [2.1]
      AW;
      L     DBW 44;	//ToASW.CmdXxxDone
      OW;
      T     DBW 44;	// --> ToASW.CmdXxxDone
NETWORK
TITLE =  auto tolerance
NX06: AN    M 197.6;	// sta_AutoTol
      JC    NX07;	// NEXT;
      L     DBW 76;	// var_AutoTolCnt
      L     DBW 188;	// par_FaultResetCntMax
      >=I;
      JC    NX07;	// NEXT;
      A     M 191.5;	// es_underWt
      O     M 191.3;	// es_TipPulse
      O     M 191.2;	// es_DosingMon
      S     M 187.7;	// cmd_retry
      JC    DOXX;
      AN    M 191.6;	// es_overWt
      JC    NX07;	// NEXT;
      L     DBD 360;	// par_TolAutoPos
      T     DBD 392;
      JCN   Y000;
      L     W#16#C;
      UC    "CWA_ScaleCtrlSub";	// S.Tolerance
Y000: A     M 199.0;	// faultPos
      O     M 199.1;	// faultNeg
      JC    NX07;	// NEXT;
      S     M 186.0;	// --> cmd_acceptWt
DOXX: L     DBW 76;	// var_AutoTolCnt
      +     1;
      T     DBW 76;	// --> var_AutoTolCnt
NETWORK
TITLE =  ALL STATE
NX07: A     M 191.0;	// EsEmpty
//[2.9]      O     M    191.1                  // EsEmptying
      O     M 191.6;	// EsOverWt
//[2.9]      O     M    191.7                  // EsZeroTol
      A     M 186.0;	// Cmd_acceptWt
      O     M 186.1;	// cmd_abortBatch
      S     M 186.2;	// --> cmd_abortIngr
      S     M 186.0;	// --> cmd_acceptWt
// 
      A     M 182.5;	// inf_closed  
      O     DBX 7.1;	// par_NoDischarging
      A     M 182.1;	// inf_enableDosingSection
      A     M 182.2;	// inf_enableDosingGrp
      AN    M 197.2;	// sta_FeedOff
      AN    M 190.2;	// EsReading
      AN    M 182.3;	// InpRefillReq
      =     M 189.2;	// --> var_enableDosing
      L     DBD 254;	// inf_ScaleWt
      L     DBD 180;	// par_EmptyWt
      <=D;
      =     M 180.4;	// --> outp_scaleEmpty
      L     MW 190;	// fault[31..00]
      L     0;
      <>I;
      JC    J1;
      T     DBW 246;	// --> errCodeSW
J1:   L     DBD 312;	// Ingr.WtActual
      L     DBD 308;	// Ingr.WtTarget
      -D;
      T     DBD 316;	// --> Ingr.WtDiff
      AN    M 189.7;	// inf_TaraSet
      JC    NX08;	// NEXT;
      L     DBD 254;	// inf_ScaleWt
      L     DBD 324;	// Ingr.PartWtTara
      AN    DBX 7.0;	// par_NegWeighing
      JC    P1;
      TAK;
P1:   -D;
      L     DBD 86;	// var_partWtByStart
      +D;
      T     DBD 312;	// --> Ingr.WtActual
NETWORK
TITLE =  ST_INIT (0000H)
NX08: L     W#16#0;	// no state
      L     DBW 240;
      <>I;
      AN    M 187.6;	// cmd_reset
      JC    NX09;	// NEXT;
      L     0;
      T     MD 192;	// --> status[47..16]
      T     DBD 42;	// --> commandsToASW
      T     MW 180;
      T     DBW 46;	// )
      T     DBD 48;	// )--> inf_activeBin[48..01]
      T     DBD 78;	// --> internalFlags
      T     MW 188;
      T     DBD 86;	// --> var_partWtByStart
      T     DBW 306;	// --> Ingr.Bin           [1G]
      T     DBD 308;	// --> Ingr.WtTarget      [1G]
      T     DBD 312;	// --> Ingr.WtActual      [1G]
      T     DBD 316;	// --> Ingr.WtDiff        [1G]
      T     DBD 320;	// --> Ingr.PartWtTarget  [1G]
      T     DBD 324;	// --> Ingr.PartWtTara    [1G]
      T     DBW 328;	// --> Ingr.DosingTime    [1G]
      L     W#16#1000;	// st_passive
      T     DBW 240;
NETWORK
TITLE =  ST_PASSIVE (1000H)
NX09: L     W#16#1000;
      L     DBW 240;
      <>I;
      JC    NX10;	// NEXT;
      R     M 181.7;	// --> inf_scaleActive
      R     M 186.2;	// --> cmd_abortIngr
      R     M 186.1;	// --> cmd_abortBatch
      R     M 196.1;	// --> sta_ScrapBatch
      L     MW 190;	// Fault
      L     2#110000000000;
      AW;
      T     MW 190;	// Fault
// 
      AN    DBX 125.2;	// ParPulseInterruptCall [1.11]
      AN    DBX 125.3;	// ParPulseTimeCall  [1.11]
      ON    DBX 7.1;	// par_NoDischarging [**1I**]
      JC    INIT;
      L     0;
      T     DBD 148;	// --> var_scale_value_input
      T     DBD 254;	// inf_ScaleWt [**1.9**]
INIT: A     M 184.0;	// cmd_readyForRecipe
      AN    M 197.3;	// sta_hold
      =     M 181.0;	// --> inf_recipeReq
      A     M 197.0;	// sta_SingleIngrMode
      A     M 184.1;	// cmd_readyForSingle(ingr)
      =     M 195.0;	// sta_SingleIngrReq
      AN    "SYS_Tick1s";
      JC    JLX;
      L     DBW 286;
      +     1;
      JO    JLX;
      T     DBW 286;	// --> inactiveTime
JLX:  A     M 183.0;	// cmd_startRecipe
      JC    T2X;	// --> st_recipe_test
      A     M 187.0;	// cmd_StartSingleIngr.
      O     M 188.2;	// cmd_SingleIngrReady
      JC    T3XX;
      JC    NX10;	// == Trans. ==
T2X:  R     M 184.0;	// --> cmd_readyForRecipe
      R     M 181.0;	// --> inf_recipeReq
      R     M 183.0;	// --> cmd_startRecipe
      S     M 193.0;	// --> sta_recipeActive
      L     W#16#2000;	// st_init_recipe
      JU    TRAN;
T3XX: R     M 181.0;	// --> inf_recipeReq
      L     0;	//                   [2.3] 
      T     DBD 274;	// --> TotalWtTarget [2.3]
      T     DBD 278;	// --> TotalWtActual [2.3]
      L     W#16#3000;	// st_wait_for_next
TRAN: T     DBW 240;	// --> st_x
      S     M 181.7;	// --> inf_scaleActive
      L     0;
      T     DBW 76;	// --> var_AutoTolCnt
NETWORK
TITLE =  ST_TEST_RECIPE (2X00H)
NX10: L     W#16#2000;
      L     DBW 240;
      ==I;
      JC    S20X;
      L     W#16#2100;	// Substate:st_recipe_test.1
      <>I;
      JC    NX11;	// == Substate 2100H ==
      A     M 186.0;	// cmd_acceptWt
      O     M 187.7;	// cmd_retry
      R     M 191.7;	// --> es_zeroTol
      JC    S20X;	// --> test again
      JU    NX11;	// == State 2000H  ==
S20X: L     0;
      T     DBD 274;	// --> TotalWtTarget
      T     DBD 278;	// --> TotalWtActual
      T     DBW 288;	// --> inf_DosingTimeBatch
      T     DBW 290;	// --> inf_WaitingForEmptying
      T     DBW 292;	// --> IngrCnt (actual)
      L     DBD 254;	// inf_ScaleWt
      T     DBD 282;	// --> TaraWtBatch
      A     M 186.1;	// cmd_abortBatch
      JC    T300;	// --> st_test_ingr
      A     DBX 7.0;	// par_NegWeighing
      JC    CEC2;	// -- zero tara_test --
      L     DBD 254;	// inf_ScaleWt
      L     DBD 180;	// par_EmptyWt
      >D;
      AN    M 186.0;	// cmd_acceptWt
      S     M 191.7;	// es_zeroTol
      L     76;	// CODE: zero_tol.
      JC    ERXO;	// ->Trans. st_recipe_error
CEC2: L     DBW 70;	// inf_recipePlace
      L     DBW 102;	// par_nr_of_recipe
      >=I;
      S     M 190.4;	// --> err_cfg_fault_SPS
      L     50;	// CODE:inf_recipe_place to big
      JC    ERXO;
      L     W#16#202;
      UC    "CWA_ScaleCtrlSub";	// S.Count ingr
      L     W#16#102;
      UC    "CWA_ScaleCtrlSub";	// S.Init_result_DB
      L     W#16#401;
      UC    "CWA_ScaleCtrlSub";	// S.Test_Bin_DB
      A     M 190.4;	// err_cfg_fault_SPS
      JC    T21X;	// --> Trans. st_recipe_error
T300: L     W#16#3000;	// st_wait_for_next
      JU    TRAX;
ERXO: T     DBW 246;	// --> errCodeSW
T21X: L     W#16#2100;	// st_recipe_error
TRAX: T     DBW 240;	// --> st_x
      R     M 183.1;	// --> cmd_ReadyForNext
      R     DBX 44.1;	// --> CMD_RESULT_BATCH_DONE
NETWORK
TITLE =  ST_WAIT_FOR_NEXT (3000H)
NX11: L     W#16#3000;
      L     DBW 240;
      <>I;
      JC    NX12;
      R     M 180.0;	// --> inf_waitForAswResult
      R     M 193.2;	// --> st_SingleIngrAc
      R     M 193.1;	// --> sta_recipeingrAc
      R     M 189.7;	// --> inf_TaraSet
      R     M 186.2;	// --> cmd_abortIngr
      R     M 193.3;	// --> sta_PartIngr
      S     M 181.1;	// --> inf_waitForNext
      L     0;
      T     DBD 46;
      T     DBW 50;	// --> active_bin[xx..01]
      T     DBD 86;	// --> var_partWtByStart
      T     DBW 306;	// --> Ingr.Bin      [1G]
      T     DBD 308;	// --> Ingr.WtTarget
      T     DBD 312;	// --> Ingr.WtActual
      T     DBD 316;	// --> Ingr.WtDiff
      T     DBD 320;	// --> Ingr.PartWtTarget
      T     DBD 324;	// --> Ingr.PartWtTara
      T     DBW 328;	// --> Ingr.DosingTime
      A     M 197.0;	// sta_SingleIngrMode
      A     M 184.1;	// cmd_readyForSingle(ingr)
      A     M 183.1;	// cmd_ReadyForNext
      =     M 195.0;	// sta_SingleIngrReq
      AN    M 197.0;	// sta_SingleIngrMode
      AN    M 193.0;	// sta_recipeActive
      JC    T100;
      AN    M 183.1;	// cmd_ReadyForNext
      JC    NX12;	// 
      A     M 187.2;	// cmd_DischargeFinal
      A     M 197.0;	// sta_SingleIngrMode
      O     M 186.1;	// cmd_abortBatch
      JC    T4X;
      A     M 187.3;	// cmd_DischargeInterm
      JC    T54X;
      AN    DBX 157.7;	// inf_ReadyForNext
      A     DBX 125.4;	// par_DosingRemote
      JC    NX12;	// 
      A     M 197.5;	// sta_step
      AN    M 187.5;	// cmd_NextStep
      JC    NX12;	// 
      AN    M 197.0;	// sta_SingleIngrMode
      JC    RECI;	// ==> read recipe ingr
      A     M 187.0;	// cmd_StartSingleIngr
      JC    IDC1;
      A     M 188.2;	// cmd_SingleIngrReady
      JC    IDC2;
      JU    NX12;
// -- read recipe ingr --
RECI: S     M 193.1;	// sta_recipeingrAc
      L     DBW 292;	// IngrCnt (actual)
      L     DBW 294;	// IngrCntTotal
      >=I;
      A     DBX 7.6;	// par_DischargeFinal
      AN    M 187.2;	// cmd_DischargeFinal
      JC    WAIT;
      L     DBW 292;	// IngrCnt (actual)
      +     1;
      T     DBW 292;	// --> IngrCnt (actual)
      L     W#16#204;
      UC    "CWA_ScaleCtrlSub";	// S.Read Recipe ingr
      JU    T4X;
// -- read single_ingr--
WAIT: L     75;
      T     DBW 246;
      JU    NX12;	// NEXT;
IDC1: S     M 193.2;	// st_SingleIngrAc
      R     M 187.0;	// cmd_StartSingleIngr
      L     DBW 64;	// NextIngr.BinNr
      T     DBW 306;	// --> ingr.BinNr
      L     DBD 66;	// NextIngr.target
      JU    TARG;
IDC2: S     M 193.2;	// st_SingleIngrAc
      L     DBW 90;	// preselected_bin
      T     DBW 306;	// --> ingr.BinNr
      L     DBD 92;	// TargetValue
TARG: T     DBD 308;	// --> ingr_TargetValue
      JU    T4X;
T100: L     W#16#1000;	// st_passive
      R     M 193.0;	// --> sta_recipeActive
      JU    TR11;	// TR11;
T54X: L     W#16#5400;	// st_DischargeInterm
      JU    TR11;	// TR11;
T4X:  L     W#16#4000;	// st_TestIngr
TR11: T     DBW 240;	// --> st_x
      R     M 195.0;	// --> sta_SingleIngrReq
      R     M 183.1;	// --> cmd_ReadyForNext
      R     M 184.2;	// --> cmd_ingrOk
      R     M 183.3;	// --> cmd_GotoWaitForNext
      R     M 188.5;	// --> flag1
      R     M 188.1;	// --> cmd_ManualAddReady
      R     M 188.2;	// --> cmd_SingleIngrReady
      R     M 188.3;	// --> cmd_ModReady
      S     DBX 207.0;	// --> CBIT
      R     M 181.1;	// --> inf_waitForNext
NETWORK
TITLE =  ST_TEST_INGR (4000H)
NX12: L     W#16#4000;
      L     DBW 240;
      <>I;
      JC    NX13;
      S     M 181.3;	// --> inf_TestIngr
      R     M 183.2;	// --> cmd_ReadyForDeselect
      A     M 187.2;	// cmd_DischargeFinal
      A     M 197.0;	// sta_SingleIngrMode
      O     M 186.1;	// cmd_abortBatch
      JC    T7X;	// --> st_DischargeFinal
      AN    M 190.3;	// err_illegel_ingr
      L     W#16#402;
      CC    "CWA_ScaleCtrlSub";	// S.Read_bin_parameter
      A     M 183.3;	// cmd_GotoWaitForNext
      AN    M 190.3;	// err_illegel_ingr
      O     M 186.2;	// cmd_abortIngr
      JC    T3X;
      AN    M 184.2;	// cmd_ingrOk
      O     M 190.3;	// err_illegel_ingr
      JC    NX13;
      L     0;
      L     DBW 306;	// ingr.BinNr
      ==I;
      JC    T7XA;	// --> st_DischargeFinal
      L     -1;
      L     DBW 306;	// ingr.BinNr
      >I;
      JC    T6X;	// --> st_working_step
      L     -1;	// DischargeInterm
      ==I;
      JC    T54Y;	// --> DischargeInterm
      JU    T5X;	// == Trans. ===
T54Y: L     W#16#5400;	// st_DischargeInterm
      JU    TR12;	// TR12;
T3X:  L     W#16#3000;	// st_wait_for_next
      JU    TR12;	// TR12;
T6X:  L     W#16#6000;	// st_working_step
      JU    TR12;	// TR12;
T7XA: L     DBW 292;	// IngrCnt
      +     -1;
      T     DBW 292;	// IngrCnt
T7X:  L     W#16#7000;	// st_DischargeFinal
      R     M 193.1;	// --> sta_RecipeIngrAc
      JU    TR12;	// TR12;
T5X:  L     W#16#5000;	// st_ingr_active
TR12: T     DBW 240;	// --> st_x
      R     M 181.3;	// --> inf_TestIngr
      R     M 183.1;	// --> cmd_ReadyForNext
      R     M 183.3;	// --> cmd_workingStepDone
      R     M 183.6;	// --> cmd_GotoWaitForNext
      R     M 184.2;	// --> cmd_ingrOk
      R     M 190.3;	// --> err_illegel_ingr
      R     M 188.5;	// --> flag1
NETWORK
TITLE =  ST_INGR_ACTIVE (5000H)
NX13: L     W#16#5000;
      L     DBW 240;
      <>I;
      JC    NX14;	// NEXT;
      R     DBX 81.2;	// ->inf_FlagStopValue
      S     #tmpNewIngr;	//[2.6]
      S     DBX 81.3;	//[2.8] ->inf_FlagNewIngr
      R     M 192.1;	// ->sta_reconveying
      L     0;
      T     DBW 384;	// ->var_CntReconveying
      T     DBW 330;	// ->Ingr.SwitchOverTime
      L     W#16#5120;	// st_test_weight
      T     DBW 240;	// ->st_x
NETWORK
TITLE =  ST_TEST_WEIGHT (5120H)
NX14: L     W#16#5120;
      L     DBW 240;
      <>I;
      JC    NX15;
      R     M 192.0;	// --> sta_TestWeighment
      A     M 196.1;	// sta_ScrapBatch
      A     M 186.1;	// cmd_abortBatch
      O     M 186.2;	// cmd_abortIngr
      O     M 188.3;	// cmd_ModReady
      JC    T56X;	// --> st_registrate_ingr
      A     M 191.5;	// es_underWt                [1H]
      A     M 186.0;	// cmd_acceptWt              [1H]
      A     DBX 337.0;	// bin_type.par_manualAdd    [1H]
      JC    T56X;	// --> st_registrate_ingr
      A     M 191.6;	// es_overWt                 [1G]   
      O     M 191.5;	// es_underWt                [1G]
      AN    M 187.7;	// cmd_retry                 [1G]
      A     DBX 337.0;	// bin_type.par_manualAdd    [1G]
      JC    NX15;	//***************************[1G]
      A     DBX 337.0;	// bin_type.par_manualAdd
      AN    M 188.1;	// cmd_ManualAddReady
      JC    T51X;	// --> st_ingr_splitt
      A     M 187.7;	// cmd_retry
      A     M 191.5;	// EsUnderWt
      R     M 188.1;	// --> CmdManualAddReady
      A     M 187.7;	// cmd_retry
      R     M 191.5;	// --> EsUnderWt
      R     M 191.6;	// --> EsOverWt
      R     M 191.2;	// --> EsDosingMon
      L     W#16#402;
      CC    "CWA_ScaleCtrlSub";	// S.Read_bin_parameter
      A     M 191.3;	// es_TipPulse
      JC    NX15;	// 
      L     DBW 342;	// BIN.par_TolPosWt
      T     DBW 392;
      L     DBW 356;	// BIN.par_TolPosPc(%)
      T     DBW 394;
      L     W#16#C;
      UC    "CWA_ScaleCtrlSub";	// S.Tolerance
      A     M 191.2;	// es_DosingMon
      AN    DBX 7.7;	// par_NoSuspendMon
      AN    M 197.7;	// sta_MonitoringOff
      O     M 191.5;	// es_underWt
      O     M 191.6;	// es_overWt
      JC    NX15;	// NEXT;
      AN    M 199.2;	// ingr_done (from FB40)
T51X: L     W#16#5100;	// --> st_ingr_splitt
      JC    TR14;	// 
T56X: L     W#16#5600;	// --> st_resulting_ingr
TR14: T     DBW 240;	// --> st_x
      R     M 184.3;	// --> cmd_AswResultDone
      R     M 191.2;	// --> es_DosingMon
      R     M 191.5;	// --> es_underWt
      R     M 191.6;	// --> es_overWt
      R     M 191.3;	// --> es_TipPulse
      R     M 193.3;	// --> StaPartIngr
      R     M 188.1;	// --> CmdMaualAdd
NETWORK
TITLE =  ST_INGR_SPLITT (5100H)
NX15: L     W#16#5100;
      L     DBW 240;
      <>I;
      JC    NX16;
      L     DBW 338;	// par_SwitchOverWt_f/s
      L     0;
      >I;
      JC    N15a;
      T     DBW 338;	// par_SwitchOverWt_f/s
N15a: L     0;
      T     DBD 320;	// --> Ingr.PartWtTarget
      A     M 193.7;	// sta_StartingDelay
      L     W#16#8;
      CC    "CWA_ScaleCtrlSub";	// S.Run Startin Delay
      A     M 187.3;	// cmd_DischargeInterm
      AN    DBX 7.0;	// par_NegWeighing
      JC    T54Z;	// -->Intermeadiate Disc.
      A     DBX 7.0;	// par_NegWeighing
      A     M 182.3;	// InpRefillReq
      JC    T53X;
      A     M 193.7;	// sta_StartingDelay
      JC    NX16;	// 
      AN    M 189.2;	// var_enableDosing
      JC    T511;	// -> suspended
      L     0;	// -- Splitt --
      L     DBD 316;	// Ingr.WtDiff
      -D;
      T     #tmpValue;	// --> var_diff_value
      A     DBX 7.0;	// par_NegWeighing
      JC    NEG;	// - positiv weighing--
      L     DBD 12;	// par_ScaleCapacityWt
      L     DBD 254;	// scale_value_absolut
      -D;
      T     DBD 392;	// --> var_max_ingredient
      L     #tmpValue;	// var_diff_value
      >=D;
      JC    VALU;	// --> CASE 1:
      L     DBD 392;	// var_max_ingredient
      L     DBD 20;	// par_ingrWtMin
      <D;
      JC    T54Z;	// --> CASE 2: Intermeadiate Disc.
      JU    C4;	// --> CASE 3/CASE4
NEG:  A     M 182.3;	// inp_refillReq
      JC    T53X;	// --> refill
      L     DBD 254;	// IF scale_value_absolut
      L     DBD 180;	// par_EmptyWt
      -D;
      T     DBD 392;	// --> var_max_ingredient
      L     #tmpValue;	// var_diff_value
      >=D;
      JC    VALU;	// --> CASE 1: = ingr.diff_value
      A     M 196.0;	// sta_RestDischarge
      JC    VALU;	// --> CASE 2: = ingr.diff_value
      L     DBD 392;	// var_max_ingredient
      L     DBD 20;	// par_ingrWtMin
      <D;
      JC    T53X;	// --> CASE 3: refill
C4:   L     #tmpValue;	// var_diff_value_ingr
      L     DBD 392;	// var_max_ingredient
      -D;
      L     DBD 20;	// par_ingrWtMin
      >=D;
      JC    P3;	// --> CASE 4 (3): max_ingredient
      L     #tmpValue;	// var_value_ingr
      L     DBD 20;	// par_ingrWtMin
      -D;	// --> CASE 5 (4):
      JU    VALU;
P3:   L     DBD 392;	// var_max_ingredient
VALU: T     DBD 320;	// --> Ingr.PartWtTarget
      L     DBD 254;	// scale_value_absolut
      T     DBD 324;	// --> Ingr.PartWtTara
      L     DBD 312;	// Ingr.WtActual
      T     DBD 86;	// --> var_partWtByStart
      L     DBD 320;	// Ingr.PartWtTarget
      +D;
      L     DBD 308;	// Ingr.WtTarget
      <D;
      =     M 193.3;	// --> sta_PartIngr
      A     DBX 125.4;	// par_DosingRemote
      JC    T52X;
      JU    T55X;	// == Trans. ===
T53X: L     W#16#5300;	// st_refill
      R     M 189.7;	// --> inf_TaraSet
      JU    TR15;	// TR15;
T55X: L     W#16#5500;	// st_dos_SPS
      S     M 189.7;	// --> inf_TaraSet
      JU    TR15;	// TR15;
T52X: L     W#16#5200;	// st_dos_remote
      S     M 189.7;	// --> inf_TaraSet
      JU    TR15;	// TR15;
T54Z: L     0;
      T     DBW 384;	// --> var_CntReconveying
      L     W#16#5400;	// st_DischargeInterm
      R     M 189.7;	// --> inf_TaraSet
      S     M 193.3;	// --> sta_PartIngr
      R     M 192.1;	//[1.10:S5.2K] ->sta_reconveying
      JU    TR15;	// TR15;
T511: L     W#16#5110;	// st_suspend
TR15: T     DBW 240;	// --> st_x
NETWORK
TITLE =  ST_SUSPENDED (5110H)
NX16: L     W#16#5110;
      L     DBW 240;
      <>I;
      JC    NX17;
      AN    DBX 7.0;	// par_NegWeighing
      ON    M 182.3;	// InpRefillReq
      AN    M 189.2;	// var_enableDosing
      AN    M 187.3;	// cmd_DischargeInterm
      AN    M 186.2;	// cmd_abortIngr
      JC    NX17;
      L     0;
      T     DBW 384;	// --> var_CntReconveying
      L     W#16#5120;	// st_test_weight
      T     DBW 240;	// --> st_x
NETWORK
TITLE =  ST_DOSING_REMOTE (5200H)
NX17: L     W#16#5200;
      L     DBW 240;
      <>I;
      JC    NX18;	// NEXT;
      A     M 188.5;	// flag1
      JC    JL1;	// [- Init State --
      S     M 188.5;
      R     DBX 81.2;	// inf_FlagStopValue
      R     DBX 157.6;	// ME.cmd_done
JL1:  A     M 189.2;	// var_enableDosing
      =     M 180.7;	// --> outp_dosing
      A     DBX 157.0;	// ME.st_stoppend
      AN    M 180.7;	// outp_dosing
      O     DBX 157.6;	// ME.cmd_done
      JC    T512;
      JU    NX18;	// NEXT;
T512: L     W#16#5120;	// st_test_weight
      T     DBW 240;	// --> st_x
      R     M 180.7;	// --> outp_dosing
      R     M 188.5;	// --> flag1
      L     W#16#404;
      UC    "CWA_ScaleCtrlSub";	// S.Save_bin_parameter
NETWORK
TITLE =  ST_REFILL (5300H)
NX18: L     W#16#5300;
      L     DBW 240;
      <>I;
      JC    NX19;	// NEXT;
      A     M 188.5;	// flag1
      JC    IN18;	// -- Init State --
      S     M 188.5;
      S     M 195.4;	// --> sta_RefillReq
      R     M 188.6;	// --> flag2_state
IN18: A     M 188.6;	// flag2_state
      JC    JL2;
      L     DBD 254;	// inf_ScaleWt
      L     DBD 12;	// par_ScaleCapacityWt
      <=D;
      AN    M 182.4;	// inp_full
      AN    M 186.0;	// cmd_acceptWt
      JC    NX19;	// NEXT;
      R     M 195.4;	// --> sta_RefillReq
      S     M 188.6;	// --> flag2_state
      S     M 193.4;	// --> sta_SettlingTime
      L     S5T#0MS;
      CLR;
      SD    T [DBW 24];	// --> Reset Timer
JL2:  L     W#16#2;
      UC    "CWA_ScaleCtrlSub";	// S.Run Settling time
      AN    M 193.4;	// sta_SettlingTime
      JC    TR18;	// 
      JU    NX19;	// 
TR18: L     W#16#5100;	// st_ingr_active
      T     DBW 240;	// --> st_x
      L     0;	//[1E:S5.2H]
      T     DBW 384;	//[1E:S5.2H] --> var_CntReconveying
      R     M 192.1;	//[1E:S5.2H] ->sta_reconveying
      R     M 188.5;	// --> flag1
NETWORK
TITLE =  ST_DOSING_PLC (5500H)
NX19: L     W#16#5500;
      L     DBW 240;
      <>I;
      JC    NX20;	// NEXT;
      R     M 189.5;	// --> cmd_NoCorrCutoffWt
      A     DBX 81.3;	//[2.8] ->inf_FlagNewIngr
      =     #tmpNewIngr;	//[2.8]
      R     DBX 81.3;	//[2.8] ->inf_FlagNewIngr
      L     DBW 384;	// var_CntReconveying
      +     1;
      T     DBW 384;	// --> var_CntReconveying
      A     DBX 337.0;	// bin_type.par_manualAdd
      JC    T551;	// --> GOTO st_maunal_add.
//[2.2]--> 
      L     DBW 338;	// par_SwitchOverWt_f/s
      ITD;
      L     DBD 320;	// Ingr.PartWtTarget
      <D;
      A(;
      L     DBW 340;	// par_CutoffWt
      ITD;
      L     DBD 320;	// Ingr.PartWtTarget
      <D;
      );
      O     #tmpNewIngr;	//[2.6]
      R     DBX 81.2;	// ->inf_FlagStopValue
//<---[2.2] 
      L     DBW 340;	// par_CutoffWt
      ITD;
      L     DBD 320;	// Ingr.PartWtTarget
      >=D;
      O     M 192.1;	// sta_reconveying
      O(;
      L     DBW 384;	// var_CntReconveying
      L     30;	///[2.2]
      >I;
      );
      O;
      A     DBX 81.2;	// inf_FlagStopValue  [2.2]
      AN    #tmpNewIngr;	//[2.6]
      JC    TX40;	// --> st_reconveying
      L     0;
      L     DBD 338;	// var_cutoff_value/var_switch_over
      <>D;
      JC    X2;	// [- Test weighment -
      L     DBD 20;	// par_ingrWtMin
      L     DBD 320;	// Ingr.PartWtTarget
      SSD   1;	// div 2
      >D;
      JC    X2;
      T     DBD 320;	// --> Ingr.PartWtTarget
      S     M 193.3;	// sta_PartIngr
      S     M 192.0;	// sta_TestWeighment --]
X2:   AN    DBX 336.7;	// bin_type.par_ModeFineDosWt
      JC    X3;
      L     DBW 340;	// par_CutoffWt
      L     DBW 368;	// par_FineDosWt
      +I;
      T     DBW 338;	// par_SwitchOverWt_f/s
X3:   L     DBD 320;	// Ingr.PartWtTarget
      L     DBW 338;	// par_SwitchOverWt_f/s
      ITD;
      <D;
      =     M 189.5;	// --> cmd_NoCorrCutoffWt
      A     DBX 337.1;	// bin_type.par_1_speed
      JC    TX30;	// --> st_slow_dos
      A     M 189.5;	// cmd_NoCorrCutoffWt
      A     DBX 337.2;	// bin_type.par_2_speed
      JC    TX30;	// --> st_slow_dos
      A     M 189.5;	// cmd_NoCorrCutoffWt
      A     DBX 337.3;	// bin_type.par_frequency_convert
      JC    TX21;	// --> st_switch_over_f/s
      L     W#16#5520;	// st_fast_dos
      JU    TR19;	// TR19;
T551: L     W#16#5510;	// st_manualAdd
      JU    TR19;	// TR19;
TX21: L     W#16#5521;	// st_switch_over_f/s
      JU    TR19;	// TR19;
TX30: L     W#16#5530;	// st_slow_dos
      JU    TR19;	// TR19
TX40: S     M 189.5;	// --> cmd_NoCorrCutoffWt
      L     W#16#5540;	// st_reconveying
TR19: T     DBW 240;	// --> st_x
      S     M 189.3;	// --> inf_DelayMon
      L     0;
      T     DBW 96;	// --> var_startingTime
      T     DBW 376;	// --> var_ActualTimeStep
      T     DBW 330;	// --> Ingr.SwitchOverTime
// 
      L     DBD 324;	// Ingr.PartWtTara
      L     DBD 320;	// Ingr.PartWtTarget
      AN    DBX 7.0;	// par_NegWeighing
      JC    POS1;
      -D;
      L     DBW 340;	// par_CutoffWt
      ITD;	// (Convert 16-Bit to 32 Bit)
      +D;
      JC    DD70;
POS1: +D;
      L     DBW 340;	// par_CutoffWt
      ITD;	// (Convert 16-Bit to 32 Bit)
      -D;
DD70: T     DBD 140;	// --> ME.var_cutoff_point
// 
      L     DBD 324;	// Ingr.PartWtTara
      L     DBD 320;	// Ingr.PartWtTarget
      AN    DBX 7.0;	// par_NegWeighing
      JC    POS2;
      -D;
      L     DBW 338;	// par_SwitchOverWt_F/S
      ITD;	// (Convert 16-Bit to 32 Bit)
      +D;
      JU    DD72;
POS2: +D;
      L     DBW 338;	// par_SwitchOverWt_F/S
      ITD;	// (Convert 16-Bit to 32 Bit)
      -D;
DD72: T     DBD 144;	// --> ME.var_switch_over_value
NETWORK
TITLE =  ST_MANUAL_ADDITION (5510H)
NX20: L     W#16#5510;
      L     DBW 240;
      <>I;
      JC    NX21;	// NEXT;
      A     M 187.4;	// cmd_ManualAddReady
      S     M 188.1;	// --> cmd_ManualAddReady
      AN    M 188.1;	// --> cmd_ManualAddReady
      AN    M 187.3;	// --> CmdDischarge
      =     M 195.1;	// --> sta_ManualAddReq
      JC    NX21;	// NEXT;
      L     W#16#5550;	// ST_SETTLING
      T     DBW 240;	// --> st_x
NETWORK
TITLE =  ST_DOSING_FAST (5520H)
NX21: L     W#16#5520;
      L     DBW 240;
      <>I;
      JC    NX22;	// NEXT;
      AN    M 191.2;	// es_DosingMon
      O     DBX 7.7;	// par_NoSuspendMon
      O     M 197.7;	// sta_MonitoringOff
      =     M 180.6;	// --> outp_dosingFast
      =     M 180.7;	// --> outp_dosing
      L     DBW 364;	// par_DosingSpeedFast
      T     DBW 296;	// --> DosingSpeed
      A     M 188.5;	// flag1
      JC    JL21;	// [- Init State --
      S     M 188.5;
      R     DBX 81.2;	// inf_FlagStopValue
      L     S5T#0MS;
      CLR;
      SD    T [DBW 24];	// --> Reset Timer
      L     0;
      T     DBW 378;	// --> varMonTime  --]
      L     S5T#20S;	// 200 ms
      AN    "SYS_infLog0";
      SP    T [DBW 24];	// --> Set timer
JL21: AN    M 189.2;	// var_enableDosing
      O     M 188.3;	// cmd_ModReady
      O     M 187.3;	// cmd_DischargeInterm
      O     M 186.2;	// cmd_abortIngr
      JC    T555;	// --> settling
      AN    T [DBW 24];	// par_timer
      JC    SEC;
      L     200;	// 200 ms
      L     T [DBW 24];	// par_timer
      -I;
      JU    T1;
SEC:  AN    "SYS_Tick1s";
      O     M 191.2;	// es_DosingMon
      JC    JM21;	// JM21;
      L     DBW 376;	// var_ActualTimeStep
      +     10;
T1:   T     DBW 376;	// --> var_ActualTimeStep
JM21: A(;
      L     DBD 144;	// ME.var_switch_over_value
      L     DBD 254;	// inf_ScaleWt
      <=D;
      AN    DBX 7.0;	// par_NegWeighing
      );
      O(;
      >=D;
      A     DBX 7.0;	// par_NegWeighing
      );
      O     DBX 81.2;	// inf_FlagStopValue
      =     #tmpStopFlag;	// --> var_switch_over_point
      A     #tmpStopFlag;	// var_switch_over_point
      A     DBX 337.3;	// bin_type.par_with_frequency_conv
      JC    TY21;	// --> GOTO st_switch_over_f/s
      A     #tmpStopFlag;	// var_switch_over_point
      JC    TX22;	// --> GOTO st_pause_f/s
      A     M 189.3;	// inf_DelayMon
      L     W#16#1;
      CC    "CWA_ScaleCtrlSub";	// S.Run DelayMon
      L     W#16#4;
      UC    "CWA_ScaleCtrlSub";	// S.DosingMon
      JU    NX22;	// == Trans. ==
TX22: L     W#16#5522;	// ST_PauseFastSlow
      JU    TR21;	// TR21;
TY21: L     W#16#5521;	// ST_SWITCH_OVER_F/S
      JU    TR21;	// TR21;
      S     M 189.5;	// --> cmd_NoCorrCutoffWt-
T555: L     W#16#5550;	// ST_SETTLING
TR21: T     DBW 240;	// --> st_x
      R     M 180.6;	// --> outp_dosingFast
      R     M 180.7;	// --> outp_dosing
      R     M 189.3;	// --> inf_DelayMon
      R     M 188.5;	// --> flag1
NETWORK
TITLE =  ST_SWITCH_OVER_F/S (5521H)
NX22: L     W#16#5521;
      L     DBW 240;
      <>I;
      JC    NX23;	// NEXT;
      R     M 180.6;	// --> outp_dosingFast
      S     M 180.7;	// --> outp_dosing
      A     M 188.5;	// flag1
      JC    N22A;	// [- Init State --
      S     M 188.5;
      R     DBX 81.2;	// inf_FlagStopValue
      L     S5T#0MS;
      CLR;
      SD    T [DBW 24];	// --> Reset Timer
      L     DBD 320;	// Ingr.PartWtTarget
      L     DBW 338;	// par_SwitchOverWt_F/S
      ITD;
      >=D;
      JC    X1;	// -- Ingr.SwitchOverTime ---
      L     DBW 340;	// par_CutoffWt
      ITD;
      -D;
      DTR;
      T     #tmpValue;	//[2.8]
      L     DBD 320;	// Ingr.PartWtTarget
      L     DBW 340;	//[2.8] par_CutoffWt
      ITD;	//[2.8]
      -D;	//[2.8]
      DTR;	//[2.8]
      L     #tmpValue;	//[2.8]
      /R;	//[2.8]
      L     DBW 350;	// par_SwitchOverTime_f/s
      DTR;
      *R;
      RND;
//[2.8]  +     L#10                        // start_delay  [***]
      JU    N27B;
X1:   L     DBW 350;	// par_SwitchOverTime_f/s
N27B: ITB;
      L     W#16#1000;	// time_base 1/10s
      OW;
      AN    "SYS_infLog0";
      SP    T [DBW 24];	// --> Set Timer
//-- End Init
N22A: AN    M 189.2;	// var_enableDosing
      JC    T55B;	// --> settling
      L     DBW 350;	// par_SwitchOverTime_f/s
      L     T [DBW 24];
      T     #tmpTimer;	// --> timer_value
      -I;
      T     DBW 330;	// --> Ingr.SwitchOverTime
      ON    T [DBW 24];	// switch over time
      O     DBX 81.2;	// inf_FlagStopValue
      JC    TY30;	// --> GOTO st_slow_dos
      L     DBW 364;	// par_DosingSpeedFast
      L     DBW 366;	// par_DosingSpeedSlow
      -I;
      T     #tmpSpeed;	// --> delta_speed
      L     #tmpTimer;	// timer_value
      DTR;
      L     DBW 350;	// par_SwitchOverTime_f/s
      DTR;
      /R;
      L     #tmpSpeed;	// delta_speed
      DTR;
      *R;
      RND;
      L     DBW 366;	// par_slow_speed
      +I;
      T     DBW 296;	// --> DosingSpeed
      L     DBW 364;	// par_DosingSpeedFast  [***
      <=I;
      JC    NX23;	// NEXT;
      T     DBW 296;	// --> DosingSpeed            ]
      JU    NX23;	// == Trans. ==
TY30: L     W#16#5530;	// ST_SLOW_dos
      JU    TR22;	// TR22;
T55B: S     M 189.5;	// --> cmd_NoCorrCutoffWt-
      L     W#16#5550;	// ST_SETTLING
TR22: T     DBW 240;	// --> st_x
      R     M 180.7;	// --> outp_dosing
      R     M 188.5;	// --> flag1
NETWORK
TITLE =  ST_PAUSE_F/S (5522H)
NX23: L     W#16#5522;
      L     DBW 240;
      <>I;
      JC    NX24;	// NEXT;
      A     M 188.5;	// flag1
      JC    JL23;	//[- Init State --
      S     M 188.5;
      R     DBX 81.2;	// --> inf_FlagStopValue
      S     M 193.6;	// -->-sta_PauseFastSlow
      L     S5T#0MS;
      CLR;
      SD    T [DBW 24];	// --> Reset Timer
      L     DBW 350;	// par_SwitchOverTime_f/s
      ITB;
      L     W#16#1000;	// time_base 1/10s
      OW;
      AN    "SYS_infLog0";
      SP    T [DBW 24];	// --> Start Timer
JL23: L     DBW 350;	// par_SwitchOverTime_f/s
      L     T [DBW 24];	// timer value
      -I;
      T     DBW 330;	// --> Ingr.SwitchOverTime
      ON    T [DBW 24];	// switch over time
      ON    M 189.2;	// var_enableDosing
      JC    TR23;	// --> settling
      JU    NX24;	// == Trans. ===
TR23: L     W#16#5530;	// ST_SLOW_dos
      T     DBW 240;	// --> st_x
      R     M 188.5;	// --> flag1
      R     M 193.6;	// --> sta_PauseFastSlow
NETWORK
TITLE =  ST_SLOW_DOSING (5530H)
NX24: L     W#16#5530;
      L     DBW 240;
      <>I;
      JC    NX25;	// NEXT;
      R     M 180.6;	// --> outp_dosingFast
      AN    M 191.2;	// es_DosingMon
      O     DBX 7.7;	// par_NoSuspendMon
      O     M 197.7;	// sta_MonitoringOff
      =     M 180.7;	// --> outp_dosing
      L     DBW 366;	// par_DosingSpeedSlow
      T     DBW 296;	// --> DosingSpeed
      A     M 188.5;	// flag1
      JC    JL24;	// [- Init State --
      S     M 188.5;
      R     DBX 81.2;	// inf_FlagStopValue
      L     S5T#0MS;
      CLR;
      SD    T [DBW 24];	// --> Reset Timer
      L     0;
      T     DBW 378;	// --> var_MonTime  --]
      L     S5T#20S;	// 200 ms
      AN    "SYS_infLog0";
      SP    T [DBW 24];	// --> Set timer
JL24: AN    M 189.2;	// var_enableDosing
      O     M 188.3;	// cmd_ModReady
      O     M 187.3;	// cmd_DischargeInterm
      O     M 186.2;	// cmd_abortIngr
      JC    SETT;	// --> settling
      AN    T [DBW 24];	// --> timer stopped
      JC    SEK;	// SEK;
      L     200;	// 200 ms
      L     T [DBW 24];
      -I;
      L     DBW 350;	// par_SwitchOverTime_f/s
      +I;
      JU    T24;	// T24;
SEK:  AN    "SYS_Tick1s";
      O     M 191.2;	// es_DosingMon
      JC    JM24;	// JM24;
      L     DBW 330;	// Ingr.SwitchOverTime
      +     10;
T24:  T     DBW 330;	// --> Ingr.SwitchOverTime
JM24: A     DBX 81.2;	// inf_FlagStopValue
      JC    SETT;	// --> GOTO st_setling
      A     M 189.3;	// inf_DelayMon
      L     W#16#1;
      CC    "CWA_ScaleCtrlSub";	// S.Run Delay Mon
      L     W#16#4;
      UC    "CWA_ScaleCtrlSub";	// S.Run Dosing Mon
      JU    NX25;	// == Trans. ==
SETT: L     W#16#5550;	// ST_SETTLING
      T     DBW 240;	// --> st_x
      R     M 180.7;	// --> outp_dosing
      R     M 188.5;	// --> flag1
NETWORK
TITLE =  ST_RECONVEYING (5540H)
NX25: L     W#16#5540;
      L     DBW 240;
      <>I;
      JC    NX26;
      R     M 180.6;	// --> outp_dosingFast
      L     DBW 366;	// par_DosingSpeedSlow
      T     DBW 296;	// --> DosingSpeed
      A     M 188.5;	// flag1
      JC    JL25;	// [- Init State --
      S     M 188.5;
      L     S5T#0MS;
      CLR;
      SD    T [DBW 24];	// --> Reset Timer
      L     0;
      T     DBW 378;	// --> var_MonTime  --]
      A     M 192.1;	// sta_reconveying
      JC    JL25;
      S     M 192.1;	// --> sta_reconveying
      L     1;
      T     DBW 384;	// --> var_CntReconveying
JL25: L     DBW 384;	// var_CntReconveying
      L     DBW 190;	// par_TipPulseCntMax
      >I;
      S     M 191.3;	// --> es_TipPulse
      JC    TR25;	// --> settling
      AN    M 189.2;	// var_enableDosing
      JC    TR25;	// --> settling
      AN    "SYS_Tick1s";
      JC    T_ON;	// T_ON;
      L     DBW 376;	// var_ActualTimeStep
      +     1;
      T     DBW 376;	// --> var_ActualTimeStep
T_ON: L     DBW 352;	// par_TipPulseLen
      ITB;
      L     W#16#1000;	// Time base 1/10s
      OW;
      SD    T [DBW 24];	// --> Start Timer
      O     T [DBW 24];	// IF actual value timer
      JC    TR25;	// TR25;
      S     M 180.7;	// --> outp_dosing
      JU    NX26;	// == Trans. ===
TR25: L     W#16#5550;	// ST_SETTLING
      T     DBW 240;	// --> st_x
      R     M 180.7;	// --> outp_dosing
      R     M 188.5;	// --> flag1
NETWORK
TITLE =  ST_SETTLING_TIME (5530H)
NX26: L     W#16#5550;
      L     DBW 240;
      <>I;
      JC    NX27;	// NEXT;
      A     M 188.5;	// flag1
      JC    JL26;	// [- Init State --
      S     M 188.5;
      S     M 193.4;	// --> sta_SettlingTime
      AN    M 189.2;	// var_enableDosing
      O     M 188.3;	// cmd_ModReady
      O     M 187.3;	// cmd_DischargeInterm
      O     M 186.2;	// cmd_abortIngr
      S     M 189.5;	// --> cmd_NoCorrCutoffWt-
      L     S5T#0MS;
      CLR;
      SD    T [DBW 24];	// --> Reset Timer
JL26: A     M 193.4;	// sta_SettlingTime
      L     W#16#2;
      CC    "CWA_ScaleCtrlSub";	// S.Run Settling Time
      A     M 193.4;	// sta_SettlingTime
      JC    NX27;	// == cor. cutoff value ==
      A     M 192.1;	// sta_reconveying
      JC    TR26;
      L     W#16#B;
      UC    "CWA_ScaleCtrlSub";	// S.Corr.CuttoffWt
      L     0;
      L     DBD 338;	// var_cutoffWt/var_switchOverWt
      <>D;
      JC    SAVE;	// -- Test weighment ---
      L     1;	// minumum 1 value must be <> 0
      T     DBW 338;	// --> var_switchOverWt
SAVE: L     W#16#404;
      UC    "CWA_ScaleCtrlSub";	// S.SaveBinParameter
TR26: SET;
      R     M 188.5;	// --> flag1
      R     M 189.3;	// --> inf_DelayMon
      L     W#16#5120;	// st_test_weight
      T     DBW 240;	// --> st_x
NETWORK
TITLE =  ST_RESULTING_INGR (5600H)
NX27: L     W#16#5600;
      L     DBW 240;
      <>I;
      JC    NX28;	// NEXT;
      AN    M 184.3;	// --> cmd_AswResultDone
      =     M 180.0;	// --> inf_waitForAswResult
      JC    NX28;	// NEXT;
      A     M 188.5;	// flag1
      JC    JL27;	// JL27;
      S     M 188.5;
      R     DBX 44.2;	// --> CMD_RESULT_ingr_DONE
      A     M 197.1;	// sta_LogOn
      S     M 189.4;	// --> cmd_IngrLog
      A     DBX 9.0;	// par_ResultPerIngrr
      S     DBX 232.2;	// --> F_RESULT_ingr
      S     DBX 207.2;	// --> CBIT
      L     W#16#104;
      UC    "CWA_ScaleCtrlSub";	// S.RegistrateIngr
JL27: A     DBX 44.2;	// CMD_RESULT_ingr_DONE
      ON    DBX 9.0;	// par_ResultPerIngr
      AN    M 189.4;	// cmd_IngrLog
      JC    T57X;
      JU    NX28;
// == Transition
T57X: L     W#16#5700;	// st_deslect
      T     DBW 240;	// --> st_x
      R     M 188.5;	// --> flag1
      R     M 184.3;	// --> cmd_AswResultDone
      R     DBX 44.2;	// --> CMD_RESULT_ingr_DONE
      R     M 183.2;	// --> cmd_ReadyForDeselect
NETWORK
TITLE =  ST_DESELECT (5700H)
NX28: L     W#16#5700;
      L     DBW 240;
      <>I;
      JC    NX29;	// NEXT;
      S     M 181.2;	// inf_deselect
      R     M 189.7;	// inf_TaraSet  [2.7]
      AN    M 183.2;	// cmd_ReadyForDeselect
      JC    NX29;	// NEXT;
      A     M 188.3;	// cmd_ModReady
      JC    T58X;
      R     M 193.2;	// --> st_SingleIngrAc      [2.3]
      L     W#16#3000;	// --> st_wait_for_next
      JU    TR28;
//Transition
T58X: L     W#16#5800;	// st_modify_ingr
TR28: T     DBW 240;	// --> st_x
      R     M 181.2;	// inf_deselect
      R     M 183.1;	// --> cmd_ReadyForNext
NETWORK
TITLE =  ST_MODIFY_INGR (5800H)
NX29: L     W#16#5800;
      L     DBW 240;
      <>I;
      JC    NX30;	// NEXT;
      R     M 188.3;	// cmd_ModReady
      R     M 189.7;	// inf_TaraSet  [**1H**]
      L     DBD 308;	// Ingr.WtTarget
      L     DBD 312;	// Ingr.WtActual
      -D;
      T     DBD 308;	// --> Ingr.WtTarget
      L     W#16#208;
      UC    "CWA_ScaleCtrlSub";	// S.StModifyRecipe
      L     0;
      T     DBD 312;	// --> Ingr.WtActual
      T     DBD 320;	// --> Ingr.PartWtTarget
      T     DBD 324;	// --> Ingr.PartWtTara
      L     DBW 90;	// var_preselected_bin
      T     DBW 306;	// --> ingr.BinNr
      SET;
      R     M 184.2;	// --> cmd_ingrOk
      R     M 183.3;	// --> cmd_GotoWaitForNext
      R     M 190.3;	// --> err_illegel_ingr
      L     W#16#4000;	// st_TestIngr
      T     DBW 240;	// --> st_x
NETWORK
TITLE =  ST_WORKING_STEP (6000H)
NX30: L     W#16#6000;
      L     DBW 240;
      <>I;
      JC    NX31;	// NEXT;
      AN    M 183.6;	// cmd_workingStepDone
      =     M 181.6;	// --> inf_workingStep
      JC    NX31;	// NEXT;
      L     W#16#3000;	// ST_WAIT_FOR_NEXT
      T     DBW 240;	// --> st_x
NETWORK
TITLE =  ST_XXXX_DISCHARGE (XXXXH)
//Segment for State:
//==================
//  7000H Main State 'st_final_discharge'
//  7010H Substate   'st_final_discharge.closing_delay'
//  7020H Substate   'st_final_discharge.start_delay'
//
//  5400H Main State 'st_intermediate_discharge'
//  5410H Substate   'st_intermediate_discharge.closing_delay'
//  5420H Substate   'st_intermediate_discharge.start_delay'
//
//
//
NX31: L     W#16#70;	// st_final_xxx
      L     DBB 240;
      <>I;
      JC    D2;
      S     M 195.2;	// --> sta_DischargeFinal
      AN    DBX 44.1;	// CMD_RESULT_BATCH_DONE
      AN    DBX 232.1;	// F_RESULT_BATCH
      A     M 184.3;	// cmd_AswResultDone
      S     DBX 232.1;	// --> F_RESULT_BATCH
      S     DBX 207.2;	// --> CBIT
      JU    ALL;
D2:   L     W#16#54;	// st_DischargeInterm
      <>I;
      JC    NX80;	// NEXT;
      S     M 195.3;	// --> sta_DischargeInterm
ALL:  SET;	// == CONTROL EMPTYING ==
      S     M 180.5;	// --> outp_readyForDischarge
      AN    M 182.5;	// inp_closed
      S     M 188.4;	// --> inf_FlagDischarge
      A     DBX 7.1;	// par_NoDischarging
      JC    T80X;
      A     DBX 241.4;	// Substate Closing (XX10H)
      JC    SXX1;	// --> Substate Closing
      A     DBX 241.5;	// Substate Start_Delay (XX20H)
      JC    SXX2;	// --> Substate Start_delay
      AN    M 191.1;	// es_EmptyingTime
      ON    M 187.7;	// cmd_retry
      A     M 188.5;	// flag1
      JC    X31;	// X31;
      S     M 188.5;
      R     M 191.1;	// es_EmptyingTime
      L     0;
      T     DBD 376;	// --> var_emptingTime/monit.time
X31:  A     M 180.4;	// outp_scaleEmpty
      O     DBX 7.0;	// par_NegWeighing
      A     M 182.6;	// inp_open
      O;
      A     M 191.1;	// es_EmptyingTime
      A     M 186.0;	// cmd_acceptWt
      JC    TXX1;	// --> Goto Substate Closing (XX10H)
      AN    M 182.6;	// inp_open
      ON    "SYS_Tick1s";
      JC    J31;
      L     DBW 290;
      +     1;
      T     DBW 290;	// --> wait_for_EmptyingTime
J31:  A     M 182.6;	// inp_open
      L     W#16#5;
      CC    "CWA_ScaleCtrlSub";	// S.MonitoringEmpyting
      JU    NX80;	// ==Substate Closing (XX10H) ==
SXX1: L     W#16#A;
      UC    "CWA_ScaleCtrlSub";	// S.Run ClosingDelay
      AN    M 193.5;	// sta_ClosingDelay
      R     M 180.5;	// --> outp_readyForDischarge
      AN    M 193.5;	// sta_ClosingDelay
      A     M 182.5;	// inp_closed
      JC    TXX2;	// --> Goto Start Delay      (XX20H)
      JU    NX80;	// ==Substate Start_Delay(XX20H)==
SXX2: R     M 180.5;	// --> outp_readyForDischarge
      AN    M 182.5;	// inp_closed
      JC    NX80;	// NEXT;
      A     M 193.7;	// sta_StartingDelay
      L     W#16#8;
      CC    "CWA_ScaleCtrlSub";	// S.Run StartingDelay
      A     M 193.7;	// sta_StartingDelay
      JC    NX80;	// NEXT;
      L     -1;	// DischargeInterm
      L     DBW 306;	// ingr.BinNr
      ==I;
      A     M 195.3;	// sta_DischargeInterm [1F:S5.2I]
      O;
      AN    M 193.2;	// st_SingleIngrAc
      AN    M 193.1;	// sta_recipeingrAc
      A     M 195.3;	// sta_DischargeInterm
      L     W#16#3000;	// ST_WAIT_FOR_NEXT
      JC    TR31;	// --> st_ingr_active
      A     M 195.3;	// sta_DischargeInterm
      L     W#16#5100;	// ST_ingr_ACTIVE
      JC    TR31;	// --> st_ingr_active
      A     M 195.2;	// sta_DischargeFinal
      JU    T80X;	// --> st_resulting_batch
TXX1: L     W#16#10;	// Substate Closing     (XX10H)
      AN    M 195.3;	// sta_DischargeInterm
      ON    DBX 7.2;	// par_NoClosingDelay
      S     M 193.5;	// --> sta_Closing_delay
      JU    SUBS;
TXX2: L     W#16#20;	// Substate Start_Delay (XX20H)
      S     M 193.7;	// --> sta_StartingDelay
SUBS: T     DBB 241;	// --> st_x.substate
      L     S5T#0MS;
      A     "SYS_infLog0";
      SD    T [DBW 24];	// --> Reset Timer
      JU    NX80;	// NEXT;
T80X: L     W#16#8000;	// ST_RESULTING_BATCH
TR31: T     DBW 240;	// --> st_x
      SET;
      R     M 180.5;	// --> outp_readyForDischarge
      R     M 195.2;	// --> sta_DischargeFinal
      R     M 195.3;	// --> sta_DischargeInterm
      R     M 188.5;	// --> flag1
      R     M 187.3;	// --> cmd_DischargeInterm
      R     M 191.1;	// --> es_EmptyingTime
      R     M 188.4;	// --> inf_FlagDischarge
NETWORK
TITLE =  ST_RESULTING_BATCH (8000H)
NX80: L     W#16#8000;
      L     DBW 240;
      <>I;
      JC    NX33;	// 
      A     M 184.3;	// cmd_AswResultDone
      AN    DBX 44.1;	// CMD_RESULT_BATCH_DONE
      AN    DBX 232.1;	// F_RESULT_BATCH
      S     DBX 232.1;	// --> F_RESULT_BATCH
      S     DBX 207.2;	// --> CBIT
      A     DBX 44.1;	// CMD_RESULT_BATCH_DONE
      ON    M 193.0;	// sta_recipeActive
      ON    DBX 9.1;	// par_ResultPerBatch
      JC    T1XX;
      JU    NX33;	// NEXT;
T1XX: L     W#16#1000;	// st_passive
      T     DBW 240;	// --> st_x
      R     M 193.0;	// --> sta_recipeActive
      R     M 184.3;	// --> cmd_AswResultDone
      R     DBX 232.1;	// --> F_RESULT_BATCH
      L     0;
      T     DBW 286;	// --> inactiveTime
NETWORK
TITLE =  Dosing Time
NX33: AN    M 193.1;	// sta_RecipeIngrAc
      AN    M 193.2;	// sta_SingleIngrAc
      O     M 195.3;	// sta_DischargeInterm
      O     M 181.4;	// inf_fault
      ON    M 189.2;	// var_enableDosing
      ON    "SYS_Tick1s";	// es_DosingMon
      JC    NX34;	// NEXT;
      L     DBW 288;	// var_dosTime_batch
      +     1;
      T     DBW 288;	// --> var_dosTime_batch
      L     DBW 328;	// var_Ingr.DosingTime
      +     1;
      T     DBW 328;	// --> var_Ingr.DosingTime
NETWORK
TITLE =  Outputs
NX34: AN    M 187.7;	// cmd_retry
      JC    N34A;
      AN    M 191.5;	// es_underWt
      AN    M 191.3;	// es_TipPulse
      JC    F2;
      R     M 192.1;	// --> sta_reconveying
      L     0;
      T     DBW 384;	// --> var_CntReconveying
F2:   L     MW 190;	// fault[31..00]
      L     2#11000000;
      AW;
      T     MW 190;
N34A: L     MW 190;	// fault[15..00]
      L     0;
      <>I;
      =     M 181.4;	// --> inf_fault
      A     M 180.7;	// --> outp_dosing
      JC    NX35;
      L     0;
      T     DBW 296;	// --> DosingSpeed
NETWORK
TITLE =  RESET COMMANDS
NX35: A     M 187.7;	// cmd_retry
      S     DBX 156.2;	// --> ME.cmd_retry
      A     M 186.0;	// cmd_retry
      S     DBX 156.3;	// --> ME.cmd_acceptWt
      A     M 186.2;	// cmd_retry
      S     DBX 156.4;	// --> ME.cmd_AbortIngr
      L     2#1111111000001000;
      L     MW 186;	// FC[47..32]
      AW;
      T     MW 186;	// --> FC[47..32]
NETWORK
TITLE =  PC_STATE
      L     DBW 238;	// StatePC
      T     #tmpValue;
      AN    M 193.0;	// sta_recipeActive
      AN    M 193.2;	// sta_SingleIngrAc
      AN    M 195.2;	// sta_DischargeFinal  [2.3]
      AN    M 181.7;	// inf_scaleActive [2.4]
      JC    N36A;	// N36A;
      A     M 195.3;	// sta_DischargeInterm
      JC    T8;
      A     M 195.2;	// sta_DischargeFinal
      AN    M 188.4;	// inf_FlagDischarge
      JC    T20;
      A     M 195.2;	// sta_DischargeFinal
      JC    T40;
      L     W#16#8000;	// st_resulting
      L     DBW 240;
      ==I;
      JC    T80;
      A     M 181.1;	// inf_waitForNext
      O     M 191.7;	// es_zeroTol
      JC    T2;
      AN    M 189.2;	// var_enableDosing
      L     W#16#10;	// suspend
      JC    STAT;
      L     4;	// dos
      JU    STAT;
N36A: L     1;	// passive
      JU    STAT;
T2:   L     2;	// waiting
      JU    STAT;
T8:   L     8;	// i.disch.
      JU    STAT;
T20:  L     W#16#20;	// complett
      JU    STAT;
T40:  L     W#16#40;	// disch.
      JU    STAT;
T80:  L     W#16#80;	// resulting
      JU    STAT;
STAT: T     DBW 238;
      A     M 181.4;	// st_fault
      =     DBX 238.7;
      AN    M 181.4;	// st_fault
      =     DBX 238.6;	// --> ST_OK
      L     DBW 238;
      L     #tmpValue;
      <>I;
      S     DBX 207.0;	// --> CBIT
NETWORK
TITLE =  Store Flags
      A     DBX 81.2;	// inf_FlagStopValue
      AN    M 192.1;	// sta_reconveying
      R     M 180.6;	// ->outp_dosingFast
      R     M 180.7;	// ->outp_dosing
      L     MW 180;
      T     DBW 42;
      L     MD 182;
      T     DBD 54;
      L     MW 186;
      T     DBW 58;
      L     MW 188;
      T     DBW 78;
      L     MW 190;
      T     DBW 244;
      L     MD 192;
      T     DBD 248;
      L     MW 196;
      T     DBW 252;
NETWORK
TITLE =  Alarm
      A     M 189.4;	// --> cmd_IngrLog
      A     DBX 9.7;	// par_LogDirectToPC
      JC    PC;
      A     M 189.4;	// cmd_IngrLog
      R     DBX 79.4;
      JC    PROT;
      L     DBW 244;	// fault[15..00]
      L     DBW 84;	// flag_fault[15..00]
      AW;
      T     DBW 84;	// --> flag_fault[15..00]
      ==I;
      JC    NX39;
      INVI;
      AW;
      JZ    NX39;
      T     #tmpFlags;	// --> new falgs
      L     0;
      T     #tmpBit;	// format_nr
LOOP: L     #tmpFlags;	// --> new falgs
      SRW   1;
      JN    DO;
      T     #tmpFlags;	// --> new falgs
      L     #tmpBit;
      INC   1;
      T     #tmpBit;
      JU    LOOP;
DO:   AN    "SYS_infLog0";
      S     DBX 43.5;	// --> cmd_horn_on
      S     DBX 207.0;	// --> CBIT
      L     #tmpBit;
      L     1;
      SLW;
      T     #tmpFlagShift;
      L     DBW 84;	// flag_fault[15..00]
      OW;
      T     DBW 84;	// --> flag_fault[15..00]
      L     #tmpBit;
      +     16;	// first msg_nr
      +     32;	// class =error
      T     DBB 391;	// --> format_nr
      L     #tmpFlagShift;
      L     2#10000010;	// es_zeroTol or es_EmptyingTime [1.8]
      AW;
      JZ    P2;
      L     DBD 254;	// scale_value
      T     MD 190;
      L     DBD 180;	// par_EmptyWt
      T     DBD 394;
      JU    LOG;
PROT: L     159;	// class=info,format=31
      T     DBB 391;	// --> format_nr
P2:   L     DBD 312;	// WtActual
      T     MD 190;
      L     DBD 308;	// WtTarget
      T     DBD 394;
LOG:  L     DBB 267;	// inf_line_nr
      T     DBB 393;
      L     DBB 29;	// par_scale_nr
      T     DBB 392;
      L     DBB 31;	// par_nr_of_dec_point
      T     DBB 390;
      L     DBW 262;	// recipeNr
      T     MW 194;
      L     0;
      T     MW 196;	// not used
      CALL  "SYS_LOG_EntryQueue" (
           DBNumber                 := 5,
           Header                   := DBW 390,
           Para1                    := DBW 392,
           Para2                    := DBW 258,
           Para3                    := DBW 260,
           Para4                    := DBW 264,
           Para5                    := DBW 306,
           Para6                    := DBW 394,
           Para7                    := DBW 396,
           Para8                    := MW 190,
           Para9                    := MW 192,
           Para10                   := MW 194,
           Para11                   := MW 196);	// MESSAGE-ENTRY /  par_nr_of_dec_point ¦ format_nr /  par_scale_Nr        ¦ inf_line_nr /  JobNumber /  JobNumberAdd /  BatchNr /  Ingredient.Bin /  WtTarget ¦ par_EmptyWt /     " /  WtActual / WtScale /     " /  RecipeNr
      JU    NX39;	// 
PC:   A     DBX 44.3;
      R     DBX 44.3;	// --> cmdLogIngrDone
      R     DBX 79.4;	// --> cmd_IngrLog
      JC    NX39;	// 
      AN    DBX 232.3;	// --> F_LogIngr
      S     DBX 232.3;	// --> F_LogIngr
      S     DBX 207.0;	// --> CBIT
NETWORK
TITLE =  END
NX39: LAR2  #tmpStoreAR2;	// Restore AR2
      BE;
END_FUNCTION

